C09153=1152.454,156.527,-58.181,-178.547,6.899,148.854
C09154=1152.449,156.776,-58.203,-178.545,6.901,148.853
C09155=1152.445,157.026,-58.224,-178.541,6.903,148.853
C09156=1152.440,157.274,-58.246,-178.539,6.905,148.852
C09157=1152.435,157.543,-58.269,-178.536,6.907,148.852
C09158=1152.430,157.812,-58.293,-178.533,6.909,148.852
C09159=1152.425,158.081,-58.315,-178.530,6.911,148.851
C09160=1152.420,158.351,-58.339,-178.527,6.913,148.851
C09161=1152.415,158.599,-58.360,-178.524,6.915,148.851
C09162=1152.410,158.848,-58.382,-178.521,6.917,148.850
C09163=1152.405,159.098,-58.403,-178.519,6.919,148.850
C09164=1152.400,159.346,-58.425,-178.516,6.921,148.850
C09165=1152.396,159.595,-58.447,-178.513,6.923,148.849
C09166=1152.391,159.844,-58.469,-178.510,6.925,148.849
C09167=1152.386,160.093,-58.491,-178.508,6.927,148.849
C09168=1152.382,160.343,-58.512,-178.504,6.929,148.848
C09169=1152.377,160.592,-58.534,-178.502,6.931,148.848
C09170=1152.372,160.840,-58.555,-178.499,6.933,148.848
C09171=1152.368,161.090,-58.577,-178.497,6.935,148.847
C09172=1152.363,161.338,-58.599,-178.494,6.936,148.847
C09173=1152.359,161.588,-58.621,-178.491,6.939,148.847
C09174=1152.353,161.837,-58.642,-178.488,6.941,148.846
C09175=1152.349,162.086,-58.664,-178.486,6.943,148.846
C09176=1152.344,162.335,-58.686,-178.483,6.945,148.846
C09177=1152.339,162.584,-58.707,-178.480,6.947,148.845
C09178=1152.335,162.833,-58.729,-178.477,6.949,148.845
C09179=1152.330,163.082,-58.751,-178.474,6.951,148.845
C09180=1152.326,163.331,-58.773,-178.472,6.952,148.844
C09181=1152.321,163.579,-58.795,-178.469,6.955,148.844
C09182=1152.316,163.828,-58.817,-178.466,6.957,148.844
C09183=1152.312,164.077,-58.839,-178.464,6.959,148.843
C09184=1152.307,164.326,-58.860,-178.460,6.961,148.843
C09185=1152.303,164.575,-58.882,-178.458,6.963,148.843
C09186=1152.297,164.824,-58.905,-178.455,6.965,148.842
C09187=1152.293,165.074,-58.927,-178.453,6.967,148.842
C09188=1152.288,165.322,-58.948,-178.449,6.969,148.842
C09189=1152.284,165.572,-58.970,-178.447,6.971,148.841
C09190=1152.279,165.820,-58.992,-178.444,6.973,148.841
C09191=1152.275,166.070,-59.014,-178.442,6.975,148.841
C09192=1152.270,166.318,-59.036,-178.438,6.977,148.840
C09193=1152.265,166.568,-59.058,-178.436,6.979,148.840
C09194=1152.260,166.816,-59.081,-178.433,6.981,148.840
C09195=1152.256,167.065,-59.103,-178.430,6.983,148.839
C09196=1152.251,167.314,-59.125,-178.428,6.986,148.839
C09197=1152.247,167.563,-59.147,-178.425,6.987,148.839
C09198=1152.241,167.812,-59.169,-178.422,6.989,148.838
C09199=1152.237,168.062,-59.191,-178.419,6.992,148.838
C09200=1152.233,168.310,-59.213,-178.416,6.993,148.838
C09201=1152.228,168.559,-59.235,-178.414,6.995,148.838
C09202=1152.223,168.808,-59.258,-178.411,6.998,148.837
C09203=1152.218,169.057,-59.280,-178.408,7.000,148.837
C09204=1152.214,169.307,-59.302,-178.405,7.001,148.836
C09205=1152.210,169.555,-59.324,-178.402,7.004,148.836
C09206=1152.205,169.804,-59.347,-178.400,7.006,148.836
C09207=1152.200,170.053,-59.368,-178.397,7.008,148.836
C09208=1152.195,170.302,-59.391,-178.394,7.010,148.835
C09209=1152.190,170.551,-59.413,-178.392,7.012,148.835
C09210=1152.186,170.800,-59.436,-178.389,7.014,148.835
C09211=1152.182,171.049,-59.458,-178.386,7.016,148.834
C09212=1152.176,171.298,-59.481,-178.383,7.018,148.834
C09213=1152.172,171.547,-59.503,-178.381,7.021,148.834
C09214=1152.167,171.796,-59.524,-178.378,7.022,148.833
C09215=1152.162,172.045,-59.548,-178.375,7.025,148.833
C09216=1152.158,172.294,-59.570,-178.372,7.027,148.833
C09217=1152.154,172.542,-59.592,-178.370,7.029,148.833
C09218=1152.149,172.792,-59.615,-178.366,7.031,148.832
C09219=1152.144,173.040,-59.636,-178.364,7.033,148.832
C09220=1152.139,173.289,-59.660,-178.361,7.035,148.832
C09221=1152.135,173.539,-59.682,-178.358,7.038,148.831
C09222=1152.130,173.787,-59.704,-178.356,7.039,148.831
C09223=1152.125,174.036,-59.727,-178.353,7.041,148.831
C09224=1152.121,174.285,-59.750,-178.350,7.044,148.830
C09225=1152.116,174.534,-59.772,-178.347,7.046,148.830
C09226=1152.112,174.783,-59.795,-178.345,7.047,148.830
C09227=1152.107,175.032,-59.817,-178.341,7.050,148.829
C09228=1152.102,175.280,-59.840,-178.339,7.052,148.829
C09229=1152.097,175.530,-59.862,-178.337,7.054,148.829
C09230=1152.093,175.779,-59.885,-178.333,7.056,148.829
C09231=1152.088,176.027,-59.907,-178.331,7.058,148.828
C09232=1152.084,176.276,-59.930,-178.328,7.061,148.828
C09233=1152.079,176.526,-59.952,-178.325,7.063,148.828
C09234=1152.075,176.775,-59.976,-178.322,7.065,148.827
C09235=1152.070,177.023,-59.998,-178.319,7.067,148.827
C09236=1152.065,177.272,-60.021,-178.317,7.069,148.827
C09237=1152.060,177.522,-60.044,-178.314,7.071,148.827
C09238=1152.055,177.770,-60.066,-178.311,7.073,148.826
C09239=1152.051,178.019,-60.089,-178.309,7.076,148.826
C09240=1152.047,178.268,-60.112,-178.306,7.077,148.826
C09241=1152.042,178.518,-60.134,-178.303,7.080,148.825
C09242=1152.037,178.766,-60.157,-178.300,7.082,148.825
C09243=1152.033,179.015,-60.180,-178.297,7.084,148.825
C09244=1152.029,179.263,-60.203,-178.295,7.086,148.824
C09245=1152.024,179.513,-60.226,-178.292,7.088,148.824
C09246=1152.018,179.761,-60.249,-178.289,7.091,148.824
C09247=1152.014,180.010,-60.271,-178.286,7.093,148.824
C09248=1152.010,180.259,-60.295,-178.283,7.095,148.823
C09249=1152.005,180.508,-60.317,-178.281,7.097,148.823
C09250=1152.001,180.757,-60.340,-178.278,7.099,148.823
C09251=1151.995,181.006,-60.363,-178.275,7.102,148.822
C09252=1151.991,181.255,-60.386,-178.273,7.104,148.822
C09253=1151.987,181.504,-60.409,-178.270,7.105,148.822
C09254=1151.982,181.753,-60.432,-178.267,7.108,148.822
C09255=1151.978,182.002,-60.455,-178.264,7.110,148.821
C09256=1151.973,182.251,-60.478,-178.261,7.113,148.821
C09257=1151.968,182.499,-60.501,-178.259,7.114,148.821
C09258=1151.964,182.748,-60.524,-178.256,7.116,148.821
C09259=1151.959,182.997,-60.547,-178.253,7.119,148.820
C09260=1151.954,183.246,-60.570,-178.250,7.121,148.820
C09261=1151.949,183.516,-60.596,-178.248,7.124,148.820
C09262=1151.944,183.785,-60.620,-178.244,7.126,148.819
C09263=1151.939,184.055,-60.645,-178.242,7.128,148.819
C09264=1151.934,184.325,-60.670,-178.238,7.131,148.819
C09265=1151.930,184.574,-60.693,-178.235,7.133,148.819
C09266=1151.925,184.823,-60.716,-178.233,7.135,148.818
C09267=1151.920,185.072,-60.740,-178.230,7.137,148.818
C09268=1151.916,185.321,-60.763,-178.227,7.140,148.818
C09269=1151.911,185.570,-60.786,-178.225,7.142,148.817
C09270=1151.907,185.818,-60.809,-178.221,7.144,148.817
C09271=1151.902,186.067,-60.832,-178.219,7.146,148.817
C09272=1151.897,186.315,-60.856,-178.216,7.149,148.817
C09273=1151.893,186.564,-60.879,-178.214,7.151,148.816
C09274=1151.888,186.813,-60.903,-178.211,7.153,148.816
C09275=1151.884,187.062,-60.926,-178.208,7.155,148.816
C09276=1151.879,187.311,-60.949,-178.205,7.157,148.816
C09277=1151.875,187.560,-60.972,-178.202,7.160,148.815
C09278=1151.870,187.809,-60.996,-178.200,7.162,148.815
C09279=1151.865,188.058,-61.019,-178.197,7.165,148.815
C09280=1151.860,188.307,-61.042,-178.194,7.166,148.814
C09281=1151.856,188.555,-61.066,-178.191,7.169,148.814
C09282=1151.851,188.805,-61.090,-178.189,7.171,148.814
C09283=1151.847,189.054,-61.113,-178.186,7.173,148.814
C09284=1151.843,189.302,-61.136,-178.183,7.176,148.814
C09285=1151.838,189.551,-61.159,-178.180,7.177,148.813
C09286=1151.834,189.800,-61.183,-178.178,7.180,148.813
C09287=1151.829,190.049,-61.207,-178.175,7.182,148.813
C09288=1151.824,190.298,-61.230,-178.172,7.185,148.812
C09289=1151.819,190.546,-61.253,-178.169,7.187,148.812
C09290=1151.815,190.795,-61.277,-178.166,7.189,148.812
C09291=1151.810,191.044,-61.300,-178.164,7.191,148.812
C09292=1151.805,191.293,-61.324,-178.161,7.194,148.811
C09293=1151.801,191.542,-61.348,-178.158,7.196,148.811
C09294=1151.797,191.791,-61.372,-178.155,7.199,148.811
C09295=1151.792,192.040,-61.395,-178.152,7.200,148.811
C09296=1151.787,192.289,-61.418,-178.150,7.203,148.811
C09297=1151.783,192.537,-61.442,-178.147,7.205,148.810
C09298=1151.778,192.786,-61.466,-178.145,7.207,148.810
C09299=1151.774,193.035,-61.490,-178.141,7.210,148.810
C09300=1151.769,193.284,-61.513,-178.139,7.212,148.810
C09301=1151.764,193.533,-61.537,-178.136,7.214,148.809
C09302=1151.760,193.781,-61.561,-178.133,7.216,148.809
C09303=1151.755,194.030,-61.584,-178.130,7.219,148.809
C09304=1151.750,194.279,-61.609,-178.128,7.221,148.808
C09305=1151.745,194.528,-61.632,-178.125,7.224,148.808
C09306=1151.741,194.776,-61.656,-178.122,7.225,148.808
C09307=1151.736,195.025,-61.679,-178.120,7.228,148.808
C09308=1151.732,195.274,-61.704,-178.117,7.230,148.807
C09309=1151.727,195.523,-61.727,-178.114,7.233,148.807
C09310=1151.723,195.771,-61.751,-178.111,7.235,148.807
C09311=1151.719,196.021,-61.775,-178.109,7.238,148.807
C09312=1151.714,196.269,-61.799,-178.106,7.239,148.807
C09313=1151.709,196.519,-61.823,-178.103,7.242,148.806
C09314=1151.705,196.767,-61.847,-178.100,7.244,148.806
C09315=1151.700,197.016,-61.870,-178.097,7.247,148.806
C09316=1151.695,197.265,-61.894,-178.094,7.250,148.806
C09317=1151.691,197.513,-61.918,-178.092,7.251,148.805
C09318=1151.687,197.763,-61.942,-178.089,7.254,148.805
C09319=1151.682,198.011,-61.967,-178.086,7.256,148.805
C09320=1151.677,198.260,-61.991,-178.083,7.259,148.805
C09321=1151.673,198.509,-62.014,-178.081,7.261,148.804
C09322=1151.668,198.757,-62.038,-178.078,7.264,148.804
C09323=1151.663,199.006,-62.063,-178.075,7.265,148.804
C09324=1151.659,199.255,-62.086,-178.072,7.268,148.804
C09325=1151.655,199.504,-62.111,-178.070,7.270,148.803
C09326=1151.650,199.753,-62.135,-178.067,7.273,148.803
C09327=1151.645,200.002,-62.159,-178.064,7.275,148.803
C09328=1151.640,200.250,-62.183,-178.061,7.278,148.803
C09329=1151.636,200.499,-62.207,-178.059,7.279,148.803
C09330=1151.632,200.748,-62.231,-178.056,7.282,148.802
C09331=1151.627,200.997,-62.256,-178.053,7.285,148.802
C09332=1151.622,201.246,-62.279,-178.050,7.287,148.802
C09333=1151.618,201.494,-62.303,-178.047,7.289,148.802
C09334=1151.614,201.743,-62.328,-178.045,7.292,148.802
C09335=1151.609,201.992,-62.353,-178.042,7.294,148.801
C09336=1151.605,202.240,-62.377,-178.040,7.296,148.801
C09337=1151.600,202.489,-62.401,-178.036,7.299,148.801
C09338=1151.596,202.739,-62.425,-178.034,7.301,148.801
C09339=1151.591,202.987,-62.449,-178.031,7.303,148.800
C09340=1151.586,203.236,-62.474,-178.028,7.306,148.800
C09341=1151.582,203.484,-62.498,-178.025,7.308,148.800
C09342=1151.578,203.733,-62.522,-178.023,7.311,148.800
C09343=1151.573,203.982,-62.547,-178.020,7.313,148.799
C09344=1151.568,204.231,-62.571,-178.017,7.316,148.799
C09345=1151.563,204.479,-62.596,-178.015,7.318,148.799
C09346=1151.559,204.728,-62.620,-178.012,7.320,148.799
C09347=1151.554,204.977,-62.645,-178.009,7.323,148.799
C09348=1151.550,205.226,-62.669,-178.006,7.325,148.798
C09349=1151.546,205.475,-62.693,-178.003,7.328,148.798
C09350=1151.541,205.723,-62.718,-178.001,7.330,148.798
C09351=1151.537,205.972,-62.742,-177.998,7.333,148.798
C09352=1151.532,206.221,-62.767,-177.995,7.334,148.797
C09353=1151.528,206.470,-62.791,-177.992,7.337,148.797
C09354=1151.522,206.718,-62.816,-177.989,7.340,148.797
C09355=1151.518,206.967,-62.840,-177.987,7.342,148.797
C09356=1151.514,207.216,-62.865,-177.984,7.345,148.797
C09357=1151.509,207.465,-62.889,-177.981,7.347,148.796
C09358=1151.505,207.714,-62.914,-177.979,7.350,148.796
C09359=1151.501,207.962,-62.939,-177.975,7.352,148.796
C09360=1151.495,208.211,-62.963,-177.973,7.354,148.796
C09361=1151.491,208.460,-62.989,-177.970,7.357,148.796
C09362=1151.486,208.708,-63.013,-177.968,7.359,148.795
C09363=1151.481,208.957,-63.037,-177.965,7.362,148.795
C09364=1151.478,209.206,-63.062,-177.962,7.364,148.795
C09365=1151.472,209.476,-63.088,-177.959,7.367,148.795
C09366=1151.468,209.747,-63.115,-177.956,7.369,148.795
C09367=1151.462,210.018,-63.143,-177.953,7.372,148.795
C09368=1151.457,210.289,-63.170,-177.950,7.375,148.794
C09369=1151.453,210.536,-63.195,-177.947,7.378,148.794
C09370=1151.448,210.785,-63.219,-177.944,7.380,148.794
C09371=1151.444,211.034,-63.244,-177.942,7.382,148.794
C09372=1151.439,211.283,-63.268,-177.939,7.385,148.794
C09373=1151.435,211.532,-63.294,-177.936,7.387,148.793
C09374=1151.431,211.780,-63.318,-177.934,7.390,148.793
C09375=1151.426,212.030,-63.343,-177.930,7.392,148.793
C09376=1151.421,212.278,-63.369,-177.928,7.394,148.793
C09377=1151.417,212.527,-63.393,-177.925,7.397,148.793
C09378=1151.412,212.776,-63.418,-177.922,7.400,148.792
C09379=1151.408,213.024,-63.443,-177.920,7.402,148.792
C09380=1151.403,213.273,-63.468,-177.917,7.405,148.792
C09381=1151.399,213.521,-63.493,-177.914,7.408,148.792
C09382=1151.394,213.770,-63.518,-177.912,7.410,148.792
C09383=1151.390,214.018,-63.543,-177.908,7.412,148.791
C09384=1151.385,214.268,-63.568,-177.906,7.414,148.791
C09385=1151.381,214.516,-63.593,-177.903,7.417,148.791
C09386=1151.376,214.765,-63.618,-177.900,7.420,148.791
C09387=1151.371,215.014,-63.643,-177.898,7.422,148.791
C09388=1151.367,215.263,-63.669,-177.895,7.425,148.791
C09389=1151.363,215.510,-63.694,-177.892,7.427,148.790
C09390=1151.358,215.760,-63.719,-177.890,7.430,148.790
C09391=1151.354,216.008,-63.744,-177.886,7.432,148.790
C09392=1151.349,216.257,-63.769,-177.884,7.435,148.790
C09393=1151.345,216.506,-63.795,-177.881,7.437,148.790
C09394=1151.340,216.755,-63.819,-177.878,7.440,148.789
C09395=1151.336,217.003,-63.845,-177.875,7.443,148.789
C09396=1151.331,217.252,-63.869,-177.873,7.445,148.789
C09397=1151.327,217.501,-63.895,-177.870,7.447,148.789
C09398=1151.322,217.749,-63.920,-177.867,7.450,148.789
C09399=1151.318,217.998,-63.945,-177.865,7.452,148.789
C09400=1151.313,218.246,-63.971,-177.862,7.455,148.788
C09401=1151.309,218.495,-63.996,-177.859,7.458,148.788
C09402=1151.305,218.744,-64.021,-177.857,7.460,148.788
C09403=1151.300,218.992,-64.046,-177.853,7.463,148.788
C09404=1151.296,219.241,-64.072,-177.851,7.466,148.788
C09405=1151.291,219.489,-64.097,-177.848,7.468,148.788
C09406=1151.286,219.739,-64.123,-177.845,7.470,148.787
C09407=1151.282,219.988,-64.148,-177.842,7.473,148.787
C09408=1151.277,220.236,-64.174,-177.839,7.476,148.787
C09409=1151.273,220.485,-64.199,-177.837,7.478,148.787
C09410=1151.268,220.734,-64.224,-177.834,7.481,148.787
C09411=1151.264,220.982,-64.250,-177.831,7.484,148.786
C09412=1151.259,221.231,-64.276,-177.829,7.486,148.786
C09413=1151.255,221.479,-64.301,-177.826,7.488,148.786
C09414=1151.250,221.728,-64.327,-177.823,7.491,148.786
C09415=1151.246,221.977,-64.352,-177.820,7.494,148.786
C09416=1151.241,222.225,-64.377,-177.818,7.496,148.786
C09417=1151.237,222.474,-64.403,-177.815,7.499,148.785
C09418=1151.233,222.723,-64.429,-177.812,7.502,148.785
C09419=1151.228,222.971,-64.454,-177.810,7.504,148.785
C09420=1151.223,223.220,-64.480,-177.806,7.506,148.785
C09421=1151.219,223.469,-64.506,-177.804,7.509,148.785
C09422=1151.214,223.717,-64.531,-177.801,7.512,148.785
C09423=1151.210,223.966,-64.557,-177.799,7.514,148.785
C09424=1151.206,224.214,-64.582,-177.795,7.517,148.784
C09425=1151.202,224.463,-64.608,-177.793,7.520,148.784
C09426=1151.197,224.711,-64.634,-177.790,7.523,148.784
C09427=1151.193,224.960,-64.659,-177.787,7.525,148.784
C09428=1151.188,225.209,-64.686,-177.784,7.528,148.784
C09429=1151.183,225.457,-64.711,-177.782,7.530,148.784
C09430=1151.179,225.706,-64.737,-177.779,7.533,148.784
C09431=1151.174,225.955,-64.763,-177.776,7.535,148.783
C09432=1151.170,226.204,-64.788,-177.773,7.538,148.783
C09433=1151.165,226.452,-64.814,-177.771,7.541,148.783
C09434=1151.161,226.701,-64.839,-177.768,7.543,148.783
C09435=1151.156,226.950,-64.866,-177.765,7.546,148.783
C09436=1151.152,227.199,-64.892,-177.762,7.549,148.783
C09437=1151.148,227.446,-64.918,-177.760,7.552,148.782
C09438=1151.143,227.695,-64.943,-177.757,7.555,148.782
C09439=1151.139,227.944,-64.969,-177.754,7.556,148.782
C09440=1151.134,228.193,-64.995,-177.751,7.559,148.782
C09441=1151.130,228.442,-65.021,-177.749,7.562,148.782
C09442=1151.125,228.690,-65.047,-177.746,7.565,148.782
C09443=1151.121,228.938,-65.073,-177.743,7.567,148.781
C09444=1151.116,229.187,-65.099,-177.740,7.570,148.781
C09445=1151.112,229.436,-65.125,-177.737,7.573,148.781
C09446=1151.108,229.685,-65.151,-177.735,7.576,148.781
C09447=1151.103,229.932,-65.177,-177.732,7.578,148.781
C09448=1151.098,230.181,-65.203,-177.729,7.580,148.781
C09449=1151.094,230.430,-65.229,-177.726,7.583,148.781
C09450=1151.090,230.679,-65.255,-177.724,7.586,148.781
C09451=1151.085,230.927,-65.282,-177.721,7.589,148.781
C09452=1151.081,231.176,-65.308,-177.719,7.591,148.780
C09453=1151.076,231.424,-65.333,-177.715,7.594,148.780
C09454=1151.071,231.673,-65.360,-177.713,7.597,148.780
C09455=1151.067,231.921,-65.386,-177.710,7.600,148.780
C09456=1151.063,232.170,-65.412,-177.708,7.602,148.780
C09457=1151.058,232.419,-65.439,-177.705,7.605,148.780
C09458=1151.054,232.668,-65.464,-177.702,7.607,148.779
C09459=1151.050,232.916,-65.491,-177.699,7.610,148.779
C09460=1151.045,233.165,-65.517,-177.696,7.613,148.779
C09461=1151.041,233.412,-65.543,-177.694,7.615,148.779
C09462=1151.036,233.661,-65.570,-177.691,7.618,148.779
C09463=1151.032,233.910,-65.596,-177.688,7.621,148.779
C09464=1151.028,234.158,-65.622,-177.685,7.624,148.779
C09465=1151.023,234.407,-65.649,-177.682,7.627,148.779
C09466=1151.019,234.656,-65.675,-177.680,7.629,148.779
C09467=1151.014,234.904,-65.702,-177.677,7.632,148.778
C09468=1151.010,235.153,-65.728,-177.674,7.635,148.778
C09469=1151.005,235.425,-65.757,-177.671,7.637,148.778
C09470=1151.000,235.697,-65.785,-177.668,7.640,148.778
C09471=1150.995,235.968,-65.814,-177.665,7.644,148.778
C09472=1150.990,236.240,-65.844,-177.662,7.646,148.778
C09473=1150.986,236.489,-65.869,-177.659,7.649,148.778
C09474=1150.981,236.737,-65.896,-177.657,7.651,148.777
C09475=1150.977,236.985,-65.923,-177.654,7.654,148.777
C09476=1150.972,237.234,-65.949,-177.651,7.657,148.777
C09477=1150.968,237.483,-65.976,-177.648,7.660,148.777
C09478=1150.963,237.731,-66.003,-177.646,7.663,148.777
C09479=1150.959,237.980,-66.029,-177.642,7.666,148.777
C09480=1150.955,238.228,-66.056,-177.640,7.668,148.777
C09481=1150.951,238.477,-66.082,-177.637,7.671,148.777
C09482=1150.946,238.726,-66.108,-177.635,7.674,148.777
C09483=1150.941,238.974,-66.135,-177.632,7.677,148.777
C09484=1150.937,239.222,-66.162,-177.629,7.680,148.776
C09485=1150.932,239.471,-66.189,-177.626,7.683,148.776
C09486=1150.928,239.719,-66.215,-177.624,7.684,148.776
C09487=1150.924,239.968,-66.242,-177.621,7.687,148.776
C09488=1150.919,240.217,-66.269,-177.618,7.690,148.776
C09489=1150.916,240.465,-66.296,-177.615,7.693,148.776
C09490=1150.911,240.714,-66.323,-177.613,7.696,148.776
C09491=1150.906,240.962,-66.350,-177.610,7.699,148.776
C09492=1150.902,241.211,-66.376,-177.607,7.702,148.776
C09493=1150.897,241.460,-66.403,-177.605,7.704,148.775
C09494=1150.893,241.708,-66.430,-177.602,7.707,148.775
C09495=1150.889,241.956,-66.456,-177.599,7.710,148.775
C09496=1150.884,242.205,-66.483,-177.596,7.712,148.775
C09497=1150.879,242.453,-66.510,-177.593,7.715,148.775
C09498=1150.876,242.702,-66.537,-177.590,7.718,148.775
C09499=1150.871,242.950,-66.564,-177.588,7.721,148.775
C09500=1150.866,243.199,-66.591,-177.585,7.723,148.775
C09501=1150.862,243.448,-66.618,-177.583,7.726,148.775
C09502=1150.858,243.696,-66.645,-177.580,7.729,148.775
C09503=1150.854,243.944,-66.672,-177.577,7.732,148.774
C09504=1150.849,244.193,-66.699,-177.574,7.735,148.774
C09505=1150.844,244.441,-66.726,-177.571,7.738,148.774
C09506=1150.840,244.690,-66.753,-177.568,7.741,148.774
C09507=1150.836,244.938,-66.779,-177.565,7.744,148.774
C09508=1150.831,245.187,-66.807,-177.563,7.746,148.774
C09509=1150.827,245.436,-66.834,-177.560,7.749,148.774
C09510=1150.822,245.684,-66.861,-177.558,7.751,148.774
C09511=1150.818,245.933,-66.888,-177.555,7.754,148.774
C09512=1150.814,246.180,-66.915,-177.552,7.757,148.774
C09513=1150.809,246.429,-66.942,-177.549,7.760,148.774
C09514=1150.805,246.678,-66.970,-177.547,7.763,148.773
C09515=1150.801,246.927,-66.997,-177.544,7.766,148.773
C09516=1150.796,247.175,-67.024,-177.541,7.769,148.773
C09517=1150.791,247.424,-67.051,-177.539,7.771,148.773
C09518=1150.787,247.671,-67.079,-177.536,7.774,148.773
C09519=1150.782,247.920,-67.106,-177.533,7.777,148.773
C09520=1150.778,248.169,-67.133,-177.530,7.780,148.773
C09521=1150.774,248.417,-67.160,-177.528,7.783,148.773
C09522=1150.770,248.665,-67.187,-177.525,7.786,148.773
C09523=1150.765,248.914,-67.215,-177.522,7.789,148.773
C09524=1150.761,249.163,-67.242,-177.519,7.792,148.773
C09525=1150.757,249.411,-67.269,-177.517,7.795,148.773
C09526=1150.752,249.659,-67.297,-177.513,7.797,148.772
C09527=1150.748,249.908,-67.324,-177.511,7.799,148.772
C09528=1150.744,250.157,-67.351,-177.508,7.802,148.772
C09529=1150.739,250.405,-67.379,-177.506,7.805,148.772
C09530=1150.735,250.653,-67.406,-177.503,7.808,148.772
C09531=1150.730,250.901,-67.434,-177.500,7.811,148.772
C09532=1150.726,251.150,-67.461,-177.497,7.814,148.772
C09533=1150.722,251.399,-67.488,-177.494,7.817,148.772
C09534=1150.717,251.647,-67.516,-177.492,7.820,148.772
C09535=1150.713,251.896,-67.544,-177.489,7.823,148.772
C09536=1150.709,252.144,-67.571,-177.486,7.826,148.772
C09537=1150.704,252.392,-67.598,-177.483,7.829,148.772
C09538=1150.700,252.640,-67.626,-177.481,7.832,148.771
C09539=1150.696,252.889,-67.654,-177.478,7.835,148.771
C09540=1150.691,253.138,-67.682,-177.475,7.838,148.771
C09541=1150.686,253.386,-67.709,-177.473,7.840,148.771
C09542=1150.682,253.635,-67.737,-177.470,7.843,148.771
C09543=1150.678,253.883,-67.764,-177.467,7.845,148.771
C09544=1150.673,254.131,-67.792,-177.464,7.848,148.771
C09545=1150.669,254.380,-67.819,-177.462,7.851,148.771
C09546=1150.665,254.628,-67.847,-177.459,7.855,148.771
C09547=1150.661,254.877,-67.875,-177.457,7.858,148.771
C09548=1150.656,255.126,-67.903,-177.454,7.860,148.771
C09549=1150.651,255.373,-67.931,-177.451,7.863,148.771
C09550=1150.647,255.623,-67.958,-177.448,7.866,148.771
C09551=1150.643,255.870,-67.986,-177.445,7.869,148.771
C09552=1150.639,256.118,-68.014,-177.443,7.872,148.771
C09553=1150.635,256.368,-68.041,-177.440,7.875,148.771
C09554=1150.629,256.616,-68.070,-177.437,7.878,148.771
C09555=1150.626,256.864,-68.098,-177.434,7.881,148.771
C09556=1150.621,257.113,-68.125,-177.432,7.884,148.770
C09557=1150.617,257.361,-68.153,-177.429,7.887,148.770
C09558=1150.612,257.610,-68.181,-177.426,7.890,148.770
C09559=1150.608,257.857,-68.209,-177.423,7.893,148.770
C09560=1150.604,258.107,-68.237,-177.420,7.896,148.770
C09561=1150.599,258.355,-68.264,-177.418,7.899,148.770
C09562=1150.595,258.603,-68.293,-177.415,7.901,148.770
C09563=1150.591,258.851,-68.321,-177.413,7.904,148.770
C09564=1150.586,259.099,-68.349,-177.410,7.907,148.770
C09565=1150.581,259.349,-68.377,-177.408,7.910,148.770
C09566=1150.577,259.597,-68.404,-177.405,7.913,148.770
C09567=1150.573,259.845,-68.433,-177.402,7.916,148.770
C09568=1150.568,260.093,-68.461,-177.399,7.919,148.770
C09569=1150.565,260.342,-68.489,-177.396,7.922,148.770
C09570=1150.560,260.590,-68.517,-177.394,7.925,148.770
C09571=1150.556,260.839,-68.546,-177.391,7.928,148.770
C09572=1150.551,261.087,-68.573,-177.388,7.930,148.770
C09573=1150.547,261.360,-68.604,-177.385,7.934,148.770
C09574=1150.542,261.633,-68.635,-177.382,7.937,148.770
C09575=1150.537,261.907,-68.666,-177.379,7.940,148.770
C09576=1150.533,262.181,-68.697,-177.376,7.944,148.769
C09577=1150.528,262.429,-68.725,-177.373,7.947,148.769
C09578=1150.524,262.678,-68.754,-177.370,7.950,148.769
C09579=1150.520,262.925,-68.782,-177.368,7.953,148.770
C09580=1150.515,263.174,-68.811,-177.365,7.956,148.769
C09581=1150.511,263.422,-68.839,-177.362,7.959,148.769
C09582=1150.506,263.671,-68.867,-177.360,7.962,148.769
C09583=1150.502,263.918,-68.895,-177.357,7.965,148.769
C09584=1150.497,264.167,-68.924,-177.354,7.968,148.769
C09585=1150.493,264.415,-68.952,-177.351,7.971,148.769
C09586=1150.489,264.664,-68.980,-177.349,7.974,148.769
C09587=1150.485,264.913,-69.008,-177.346,7.977,148.769
C09588=1150.480,265.161,-69.037,-177.343,7.980,148.769
C09589=1150.476,265.409,-69.066,-177.341,7.983,148.769
C09590=1150.471,265.657,-69.094,-177.338,7.986,148.769
C09591=1150.468,265.906,-69.122,-177.335,7.989,148.769
C09592=1150.463,266.154,-69.151,-177.332,7.991,148.769
C09593=1150.459,266.402,-69.179,-177.330,7.995,148.769
C09594=1150.455,266.651,-69.208,-177.327,7.998,148.769
C09595=1150.449,266.899,-69.237,-177.324,8.001,148.769
C09596=1150.446,267.147,-69.265,-177.322,8.004,148.769
C09597=1150.441,267.396,-69.293,-177.319,8.007,148.769
C09598=1150.437,267.643,-69.322,-177.316,8.009,148.769
C09599=1150.433,267.892,-69.351,-177.314,8.013,148.769
C09600=1150.428,268.141,-69.379,-177.311,8.016,148.769
C09601=1150.424,268.388,-69.408,-177.308,8.019,148.769
C09602=1150.420,268.637,-69.437,-177.305,8.022,148.769
C09603=1150.415,268.885,-69.464,-177.303,8.024,148.769
C09604=1150.411,269.134,-69.494,-177.300,8.027,148.769
C09605=1150.407,269.382,-69.523,-177.298,8.031,148.769
C09606=1150.403,269.630,-69.551,-177.295,8.034,148.769
C09607=1150.398,269.879,-69.580,-177.292,8.037,148.769
C09608=1150.394,270.127,-69.609,-177.289,8.040,148.769
C09609=1150.390,270.375,-69.637,-177.286,8.042,148.769
C09610=1150.385,270.624,-69.666,-177.284,8.047,148.769
C09611=1150.381,270.872,-69.695,-177.281,8.049,148.769
C09612=1150.376,271.121,-69.724,-177.278,8.052,148.769
C09613=1150.372,271.368,-69.752,-177.275,8.055,148.769
C09614=1150.368,271.617,-69.781,-177.273,8.059,148.769
C09615=1150.364,271.865,-69.811,-177.270,8.062,148.769
C09616=1150.359,272.114,-69.839,-177.267,8.064,148.769
C09617=1150.355,272.361,-69.868,-177.265,8.067,148.769
C09618=1150.351,272.610,-69.897,-177.262,8.070,148.769
C09619=1150.346,272.858,-69.926,-177.260,8.074,148.769
C09620=1150.342,273.107,-69.956,-177.257,8.077,148.769
C09621=1150.338,273.355,-69.983,-177.254,8.080,148.769
C09622=1150.334,273.603,-70.013,-177.251,8.082,148.769
C09623=1150.329,273.852,-70.041,-177.249,8.086,148.769
C09624=1150.325,274.100,-70.071,-177.246,8.089,148.769
C09625=1150.320,274.348,-70.100,-177.243,8.092,148.769
C09626=1150.316,274.596,-70.129,-177.241,8.095,148.769
C09627=1150.312,274.844,-70.158,-177.238,8.099,148.769
C09628=1150.308,275.093,-70.187,-177.235,8.102,148.769
C09629=1150.304,275.341,-70.217,-177.232,8.105,148.769
C09630=1150.299,275.589,-70.245,-177.229,8.107,148.769
C09631=1150.295,275.837,-70.274,-177.227,8.111,148.769
C09632=1150.291,276.086,-70.304,-177.224,8.114,148.769
C09633=1150.286,276.334,-70.333,-177.221,8.117,148.769
C09634=1150.282,276.583,-70.362,-177.219,8.120,148.769
C09635=1150.278,276.831,-70.391,-177.216,8.123,148.769
C09636=1150.274,277.078,-70.420,-177.214,8.126,148.769
C09637=1150.269,277.327,-70.449,-177.211,8.129,148.769
C09638=1150.265,277.575,-70.479,-177.208,8.132,148.769
C09639=1150.261,277.824,-70.508,-177.206,8.135,148.769
C09640=1150.257,278.072,-70.537,-177.202,8.139,148.769
C09641=1150.252,278.320,-70.566,-177.200,8.142,148.769
C09642=1150.248,278.569,-70.596,-177.197,8.145,148.769
C09643=1150.244,278.817,-70.625,-177.194,8.148,148.769
C09644=1150.239,279.064,-70.654,-177.192,8.151,148.769
C09645=1150.235,279.313,-70.684,-177.189,8.154,148.769
C09646=1150.231,279.561,-70.713,-177.187,8.157,148.769
C09647=1150.227,279.809,-70.743,-177.184,8.160,148.769
C09648=1150.223,280.057,-70.772,-177.182,8.163,148.769
C09649=1150.218,280.306,-70.802,-177.179,8.166,148.769
C09650=1150.214,280.554,-70.831,-177.175,8.170,148.769
C09651=1150.210,280.802,-70.861,-177.173,8.173,148.769
C09652=1150.206,281.051,-70.890,-177.170,8.176,148.769
C09653=1150.201,281.299,-70.920,-177.168,8.179,148.769
C09654=1150.197,281.547,-70.950,-177.165,8.182,148.769
C09655=1150.192,281.795,-70.979,-177.162,8.185,148.769
C09656=1150.188,282.043,-71.008,-177.160,8.189,148.769
C09657=1150.184,282.292,-71.038,-177.157,8.191,148.769
C09658=1150.179,282.540,-71.067,-177.155,8.194,148.769
C09659=1150.175,282.788,-71.097,-177.152,8.198,148.770
C09660=1150.171,283.036,-71.127,-177.149,8.201,148.770
C09661=1150.166,283.284,-71.157,-177.146,8.204,148.769
C09662=1150.162,283.533,-71.186,-177.144,8.208,148.770
C09663=1150.158,283.781,-71.216,-177.141,8.211,148.770
C09664=1150.154,284.029,-71.245,-177.138,8.214,148.770
C09665=1150.150,284.277,-71.275,-177.136,8.217,148.770
C09666=1150.145,284.525,-71.305,-177.133,8.220,148.770
C09667=1150.141,284.774,-71.335,-177.130,8.224,148.770
C09668=1150.137,285.022,-71.364,-177.127,8.227,148.770
C09669=1150.133,285.270,-71.394,-177.125,8.230,148.770
C09670=1150.129,285.518,-71.424,-177.122,8.233,148.770
C09671=1150.124,285.766,-71.454,-177.120,8.236,148.770
C09672=1150.120,286.015,-71.483,-177.117,8.239,148.770
C09673=1150.116,286.262,-71.514,-177.115,8.242,148.770
C09674=1150.112,286.511,-71.543,-177.111,8.246,148.770
C09675=1150.107,286.759,-71.573,-177.109,8.249,148.770
C09676=1150.103,287.007,-71.603,-177.106,8.252,148.770
C09677=1150.098,287.283,-71.636,-177.104,8.255,148.770
C09678=1150.094,287.558,-71.669,-177.100,8.259,148.770
C09679=1150.089,287.833,-71.702,-177.097,8.263,148.770
C09680=1150.084,288.109,-71.736,-177.095,8.266,148.770
C09681=1150.080,288.357,-71.766,-177.092,8.269,148.770
C09682=1150.076,288.605,-71.796,-177.089,8.273,148.770
C09683=1150.071,288.853,-71.826,-177.086,8.276,148.771
C09684=1150.067,289.101,-71.856,-177.084,8.279,148.771
C09685=1150.063,289.349,-71.886,-177.081,8.282,148.771
C09686=1150.058,289.597,-71.916,-177.078,8.285,148.771
C09687=1150.054,289.845,-71.946,-177.076,8.289,148.771
C09688=1150.050,290.094,-71.977,-177.073,8.292,148.771
C09689=1150.046,290.342,-72.007,-177.070,8.296,148.771
C09690=1150.042,290.590,-72.037,-177.068,8.299,148.771
C09691=1150.038,290.838,-72.067,-177.065,8.302,148.771
C09692=1150.033,291.086,-72.097,-177.063,8.305,148.771
C09693=1150.029,291.334,-72.128,-177.060,8.308,148.771
C09694=1150.025,291.582,-72.157,-177.057,8.312,148.771
C09695=1150.021,291.831,-72.188,-177.054,8.315,148.771
C09696=1150.017,292.079,-72.218,-177.052,8.318,148.771
C09697=1150.012,292.327,-72.248,-177.049,8.321,148.771
C09698=1150.008,292.575,-72.279,-177.047,8.324,148.772
C09699=1150.004,292.823,-72.309,-177.044,8.327,148.772
C09700=1150.000,293.071,-72.340,-177.041,8.331,148.772
C09701=1149.996,293.320,-72.369,-177.038,8.334,148.772
C09702=1149.991,293.567,-72.400,-177.036,8.337,148.772
C09703=1149.987,293.815,-72.431,-177.033,8.340,148.772
C09704=1149.982,294.064,-72.460,-177.031,8.344,148.772
C09705=1149.978,294.312,-72.491,-177.028,8.347,148.772
C09706=1149.974,294.560,-72.522,-177.025,8.351,148.772
C09707=1149.970,294.808,-72.552,-177.022,8.354,148.772
C09708=1149.966,295.056,-72.583,-177.020,8.357,148.772
C09709=1149.962,295.305,-72.613,-177.017,8.360,148.772
C09710=1149.958,295.553,-72.643,-177.014,8.364,148.773
C09711=1149.953,295.801,-72.674,-177.012,8.367,148.773
C09712=1149.949,296.048,-72.705,-177.009,8.370,148.773
C09713=1149.945,296.297,-72.735,-177.007,8.373,148.773
C09714=1149.941,296.545,-72.766,-177.004,8.376,148.773
C09715=1149.937,296.792,-72.796,-177.001,8.381,148.773
C09716=1149.932,297.040,-72.827,-176.999,8.383,148.773
C09717=1149.928,297.289,-72.858,-176.996,8.387,148.773
C09718=1149.924,297.537,-72.888,-176.993,8.390,148.773
C09719=1149.920,297.785,-72.919,-176.991,8.393,148.773
C09720=1149.916,298.033,-72.950,-176.988,8.397,148.773
C09721=1149.912,298.281,-72.980,-176.985,8.400,148.773
C09722=1149.907,298.529,-73.011,-176.983,8.403,148.774
C09723=1149.903,298.777,-73.042,-176.980,8.406,148.774
C09724=1149.899,299.026,-73.073,-176.978,8.410,148.774
C09725=1149.895,299.273,-73.103,-176.975,8.413,148.774
C09726=1149.890,299.521,-73.134,-176.972,8.417,148.774
C09727=1149.886,299.770,-73.165,-176.970,8.420,148.774
C09728=1149.881,300.018,-73.196,-176.967,8.423,148.774
C09729=1149.878,300.265,-73.226,-176.964,8.427,148.774
C09730=1149.874,300.514,-73.257,-176.962,8.430,148.774
C09731=1149.869,300.762,-73.288,-176.959,8.433,148.774
C09732=1149.865,301.011,-73.319,-176.957,8.436,148.775
C09733=1149.861,301.258,-73.350,-176.954,8.440,148.775
C09734=1149.857,301.506,-73.381,-176.951,8.443,148.775
C09735=1149.853,301.754,-73.412,-176.949,8.446,148.775
C09736=1149.848,302.002,-73.442,-176.946,8.450,148.775
C09737=1149.844,302.250,-73.473,-176.943,8.454,148.775
C09738=1149.840,302.498,-73.505,-176.941,8.457,148.775
C09739=1149.836,302.746,-73.535,-176.938,8.460,148.775
C09740=1149.832,302.995,-73.566,-176.936,8.463,148.776
C09741=1149.827,303.243,-73.597,-176.933,8.466,148.776
C09742=1149.823,303.490,-73.629,-176.930,8.470,148.776
C09743=1149.819,303.739,-73.660,-176.927,8.473,148.776
C09744=1149.814,303.986,-73.690,-176.925,8.476,148.776
C09745=1149.811,304.235,-73.722,-176.923,8.480,148.776
C09746=1149.806,304.482,-73.753,-176.920,8.483,148.776
C09747=1149.802,304.731,-73.784,-176.917,8.487,148.776
C09748=1149.798,304.978,-73.816,-176.915,8.490,148.776
C09749=1149.793,305.226,-73.846,-176.912,8.494,148.776
C09750=1149.789,305.474,-73.878,-176.909,8.497,148.777
C09751=1149.785,305.722,-73.909,-176.907,8.500,148.777
C09752=1149.782,305.971,-73.940,-176.904,8.503,148.777
C09753=1149.777,306.218,-73.971,-176.901,8.507,148.777
C09754=1149.773,306.467,-74.002,-176.899,8.511,148.777
C09755=1149.769,306.714,-74.034,-176.896,8.514,148.777
C09756=1149.765,306.963,-74.065,-176.894,8.517,148.777
C09757=1149.761,307.210,-74.096,-176.891,8.521,148.778
C09758=1149.756,307.459,-74.128,-176.889,8.524,148.778
C09759=1149.752,307.706,-74.160,-176.886,8.527,148.778
C09760=1149.748,307.955,-74.191,-176.883,8.530,148.778
C09761=1149.743,308.202,-74.222,-176.881,8.534,148.778
C09762=1149.739,308.451,-74.253,-176.878,8.537,148.778
C09763=1149.735,308.698,-74.285,-176.875,8.541,148.778
C09764=1149.731,308.946,-74.317,-176.873,8.545,148.778
C09765=1149.727,309.194,-74.347,-176.870,8.548,148.779
C09766=1149.723,309.442,-74.379,-176.867,8.551,148.779
C09767=1149.719,309.690,-74.411,-176.865,8.554,148.779
C09768=1149.715,309.938,-74.442,-176.862,8.558,148.779
C09769=1149.711,310.186,-74.474,-176.859,8.561,148.779
C09770=1149.706,310.434,-74.506,-176.857,8.565,148.779
C09771=1149.702,310.683,-74.537,-176.854,8.569,148.779
C09772=1149.697,310.930,-74.568,-176.852,8.572,148.780
C09773=1149.694,311.178,-74.600,-176.849,8.575,148.780
C09774=1149.689,311.426,-74.631,-176.846,8.579,148.780
C09775=1149.685,311.674,-74.663,-176.844,8.582,148.780
C09776=1149.682,311.922,-74.695,-176.842,8.586,148.780
C09777=1149.677,312.170,-74.727,-176.839,8.588,148.780
C09778=1149.673,312.418,-74.759,-176.836,8.593,148.780
C09779=1149.668,312.666,-74.789,-176.834,8.596,148.781
C09780=1149.665,312.914,-74.821,-176.831,8.599,148.781
C09781=1149.660,313.191,-74.857,-176.828,8.603,148.781
C09782=1149.655,313.469,-74.893,-176.825,8.607,148.781
C09783=1149.651,313.747,-74.929,-176.822,8.611,148.781
C09784=1149.646,314.024,-74.964,-176.819,8.615,148.781
C09785=1149.642,314.272,-74.996,-176.817,8.618,148.782
C09786=1149.638,314.521,-75.027,-176.814,8.621,148.782
C09787=1149.633,314.768,-75.059,-176.811,8.625,148.782
C09788=1149.630,315.016,-75.091,-176.809,8.629,148.782
C09789=1149.625,315.264,-75.123,-176.807,8.632,148.782
C09790=1149.621,315.512,-75.155,-176.804,8.636,148.782
C09791=1149.617,315.760,-75.186,-176.801,8.639,148.783
C09792=1149.613,316.008,-75.218,-176.799,8.642,148.783
C09793=1149.609,316.256,-75.251,-176.796,8.646,148.783
C09794=1149.605,316.503,-75.282,-176.793,8.650,148.783
C09795=1149.600,316.752,-75.315,-176.791,8.653,148.783
C09796=1149.597,317.000,-75.347,-176.788,8.657,148.783
C09797=1149.593,317.247,-75.379,-176.786,8.660,148.784
C09798=1149.588,317.495,-75.411,-176.783,8.663,148.784
C09799=1149.584,317.743,-75.443,-176.780,8.667,148.784
C09800=1149.581,317.991,-75.475,-176.778,8.671,148.784
C09801=1149.576,318.239,-75.507,-176.776,8.674,148.784
C09802=1149.572,318.487,-75.539,-176.773,8.678,148.784
C09803=1149.567,318.735,-75.571,-176.770,8.681,148.785
C09804=1149.564,318.983,-75.603,-176.768,8.684,148.785
C09805=1149.560,319.230,-75.635,-176.765,8.688,148.785
C09806=1149.555,319.478,-75.668,-176.762,8.692,148.785
C09807=1149.552,319.726,-75.700,-176.760,8.695,148.785
C09808=1149.547,319.975,-75.732,-176.757,8.699,148.785
C09809=1149.544,320.222,-75.765,-176.755,8.702,148.786
C09810=1149.539,320.470,-75.797,-176.752,8.705,148.786
C09811=1149.535,320.718,-75.828,-176.750,8.710,148.786
C09812=1149.531,320.966,-75.861,-176.747,8.713,148.786
C09813=1149.527,321.213,-75.893,-176.744,8.716,148.786
C09814=1149.523,321.462,-75.926,-176.742,8.720,148.786
C09815=1149.518,321.709,-75.957,-176.739,8.723,148.787
C09816=1149.514,321.957,-75.991,-176.736,8.727,148.787
C09817=1149.511,322.205,-76.022,-176.734,8.730,148.787
C09818=1149.506,322.453,-76.056,-176.732,8.734,148.787
C09819=1149.503,322.701,-76.087,-176.729,8.738,148.788
C09820=1149.498,322.949,-76.120,-176.726,8.741,148.788
C09821=1149.494,323.196,-76.153,-176.724,8.744,148.788
C09822=1149.490,323.444,-76.184,-176.721,8.748,148.788
C09823=1149.486,323.692,-76.218,-176.719,8.752,148.788
C09824=1149.482,323.940,-76.249,-176.716,8.756,148.789
C09825=1149.478,324.188,-76.283,-176.714,8.759,148.789
C09826=1149.473,324.436,-76.315,-176.711,8.762,148.789
C09827=1149.470,324.683,-76.348,-176.708,8.766,148.789
C09828=1149.466,324.932,-76.380,-176.706,8.769,148.789
C09829=1149.461,325.179,-76.413,-176.703,8.773,148.789
C09830=1149.457,325.427,-76.445,-176.700,8.777,148.790
C09831=1149.453,325.674,-76.478,-176.698,8.780,148.790
C09832=1149.449,325.923,-76.510,-176.695,8.784,148.790
C09833=1149.445,326.170,-76.543,-176.693,8.787,148.790
C09834=1149.441,326.418,-76.576,-176.691,8.791,148.790
C09835=1149.437,326.666,-76.608,-176.688,8.795,148.791
C09836=1149.433,326.914,-76.641,-176.685,8.798,148.791
C09837=1149.429,327.162,-76.673,-176.682,8.802,148.791
C09838=1149.425,327.410,-76.707,-176.680,8.805,148.791
C09839=1149.420,327.658,-76.740,-176.678,8.809,148.791
C09840=1149.417,327.905,-76.772,-176.675,8.813,148.792
C09841=1149.413,328.153,-76.805,-176.673,8.816,148.792
C09842=1149.408,328.401,-76.838,-176.670,8.820,148.792
C09843=1149.404,328.649,-76.871,-176.667,8.823,148.792
C09844=1149.401,328.897,-76.903,-176.664,8.827,148.793
C09845=1149.396,329.145,-76.936,-176.662,8.831,148.793
C09846=1149.392,329.392,-76.969,-176.660,8.834,148.793
C09847=1149.388,329.640,-77.002,-176.657,8.838,148.793
C09848=1149.384,329.888,-77.036,-176.655,8.841,148.793
C09849=1149.380,330.136,-77.068,-176.652,8.845,148.794
C09850=1149.376,330.383,-77.101,-176.649,8.849,148.794
C09851=1149.372,330.631,-77.134,-176.647,8.852,148.794
C09852=1149.368,330.879,-77.167,-176.644,8.856,148.794
C09853=1149.364,331.127,-77.200,-176.642,8.859,148.794
C09854=1149.360,331.374,-77.233,-176.639,8.864,148.795
C09855=1149.356,331.622,-77.266,-176.637,8.867,148.795
C09856=1149.351,331.870,-77.299,-176.634,8.871,148.795
C09857=1149.347,332.118,-77.333,-176.632,8.874,148.796
C09858=1149.343,332.366,-77.365,-176.629,8.878,148.796
C09859=1149.339,332.613,-77.398,-176.626,8.882,148.796
C09860=1149.335,332.861,-77.431,-176.624,8.885,148.796
C09861=1149.331,333.109,-77.464,-176.621,8.889,148.796
C09862=1149.327,333.357,-77.497,-176.619,8.892,148.797
C09863=1149.323,333.604,-77.530,-176.616,8.896,148.797
C09864=1149.319,333.852,-77.563,-176.614,8.900,148.797
C09865=1149.315,334.099,-77.597,-176.611,8.904,148.797
C09866=1149.311,334.347,-77.630,-176.608,8.907,148.798
C09867=1149.307,334.595,-77.664,-176.607,8.911,148.798
C09868=1149.303,334.843,-77.697,-176.604,8.915,148.798
C09869=1149.299,335.091,-77.730,-176.601,8.918,148.798
C09870=1149.295,335.338,-77.763,-176.598,8.922,148.799
C09871=1149.291,335.586,-77.797,-176.596,8.925,148.799
C09872=1149.287,335.834,-77.830,-176.593,8.929,148.799
C09873=1149.283,336.081,-77.864,-176.591,8.933,148.799
C09874=1149.279,336.329,-77.897,-176.588,8.937,148.799
C09875=1149.275,336.577,-77.930,-176.586,8.940,148.800
C09876=1149.270,336.825,-77.964,-176.583,8.944,148.800
C09877=1149.266,337.073,-77.997,-176.581,8.948,148.800
C09878=1149.262,337.320,-78.031,-176.578,8.952,148.801
C09879=1149.258,337.568,-78.064,-176.576,8.955,148.801
C09880=1149.254,337.815,-78.097,-176.573,8.958,148.801
C09881=1149.250,338.064,-78.131,-176.570,8.962,148.801
C09882=1149.247,338.311,-78.165,-176.568,8.966,148.801
C09883=1149.242,338.559,-78.198,-176.566,8.970,148.802
C09884=1149.238,338.807,-78.232,-176.563,8.973,148.802
C09885=1149.234,339.087,-78.270,-176.560,8.978,148.802
C09886=1149.229,339.367,-78.307,-176.557,8.982,148.803
C09887=1149.224,339.647,-78.346,-176.554,8.987,148.803
C09888=1149.220,339.928,-78.383,-176.552,8.991,148.803
C09889=1149.216,340.175,-78.418,-176.549,8.994,148.804
C09890=1149.211,340.423,-78.451,-176.546,8.998,148.804
C09891=1149.207,340.670,-78.484,-176.544,9.002,148.804
C09892=1149.204,340.918,-78.519,-176.541,9.006,148.804
C09893=1149.199,341.166,-78.552,-176.539,9.009,148.804
C09894=1149.195,341.413,-78.586,-176.536,9.013,148.805
C09895=1149.191,341.661,-78.619,-176.534,9.017,148.805
C09896=1149.188,341.909,-78.654,-176.531,9.021,148.805
C09897=1149.183,342.157,-78.687,-176.529,9.024,148.806
C09898=1149.179,342.404,-78.721,-176.526,9.028,148.806
C09899=1149.175,342.652,-78.754,-176.524,9.032,148.806
C09900=1149.171,342.900,-78.789,-176.521,9.036,148.806
C09901=1149.167,343.147,-78.823,-176.519,9.039,148.807
C09902=1149.163,343.395,-78.856,-176.516,9.043,148.807
C09903=1149.159,343.642,-78.891,-176.514,9.047,148.807
C09904=1149.155,343.891,-78.924,-176.511,9.051,148.808
C09905=1149.151,344.138,-78.958,-176.509,9.054,148.808
C09906=1149.147,344.385,-78.992,-176.506,9.058,148.808
C09907=1149.143,344.634,-79.026,-176.504,9.062,148.808
C09908=1149.139,344.881,-79.060,-176.501,9.066,148.809
C09909=1149.135,345.128,-79.094,-176.499,9.069,148.809
C09910=1149.131,345.377,-79.128,-176.496,9.073,148.809
C09911=1149.127,345.624,-79.162,-176.494,9.077,148.809
C09912=1149.123,345.871,-79.196,-176.491,9.081,148.810
C09913=1149.119,346.119,-79.231,-176.489,9.084,148.810
C09914=1149.115,346.366,-79.265,-176.486,9.088,148.810
C09915=1149.111,346.614,-79.298,-176.483,9.093,148.811
C09916=1149.107,346.862,-79.333,-176.481,9.096,148.811
C09917=1149.103,347.109,-79.367,-176.478,9.100,148.811
C09918=1149.099,347.357,-79.402,-176.476,9.103,148.812
C09919=1149.095,347.605,-79.435,-176.473,9.108,148.812
C09920=1149.090,347.853,-79.469,-176.471,9.111,148.812
C09921=1149.087,348.100,-79.503,-176.468,9.115,148.812
C09922=1149.083,348.348,-79.538,-176.466,9.119,148.813
C09923=1149.079,348.596,-79.572,-176.463,9.123,148.813
C09924=1149.075,348.843,-79.607,-176.461,9.126,148.813
C09925=1149.071,349.090,-79.641,-176.458,9.130,148.814
C09926=1149.067,349.338,-79.675,-176.455,9.134,148.814
C09927=1149.063,349.585,-79.709,-176.453,9.138,148.814
C09928=1149.059,349.833,-79.744,-176.451,9.142,148.814
C09929=1149.055,350.081,-79.779,-176.448,9.145,148.815
C09930=1149.051,350.329,-79.813,-176.445,9.149,148.815
C09931=1149.047,350.576,-79.847,-176.443,9.153,148.815
C09932=1149.043,350.823,-79.881,-176.441,9.157,148.816
C09933=1149.039,351.071,-79.916,-176.438,9.160,148.816
C09934=1149.035,351.319,-79.950,-176.436,9.165,148.816
C09935=1149.031,351.567,-79.985,-176.433,9.169,148.817
C09936=1149.027,351.814,-80.019,-176.430,9.172,148.817
C09937=1149.023,352.062,-80.053,-176.428,9.176,148.817
C09938=1149.019,352.309,-80.089,-176.426,9.180,148.817
C09939=1149.015,352.557,-80.123,-176.423,9.184,148.818
C09940=1149.011,352.804,-80.157,-176.420,9.188,148.818
C09941=1149.007,353.052,-80.192,-176.418,9.192,148.818
C09942=1149.003,353.299,-80.227,-176.415,9.196,148.819
C09943=1149.000,353.547,-80.261,-176.413,9.199,148.819
C09944=1148.995,353.794,-80.296,-176.410,9.203,148.819
C09945=1148.991,354.042,-80.331,-176.408,9.207,148.819
C09946=1148.987,354.290,-80.365,-176.405,9.211,148.820
C09947=1148.984,354.537,-80.399,-176.403,9.215,148.820
C09948=1148.980,354.785,-80.435,-176.401,9.219,148.821
C09949=1148.975,355.032,-80.469,-176.398,9.223,148.821
C09950=1148.972,355.280,-80.504,-176.395,9.226,148.821
C09951=1148.968,355.527,-80.539,-176.393,9.230,148.822
C09952=1148.964,355.775,-80.574,-176.390,9.234,148.822
C09953=1148.959,356.022,-80.608,-176.388,9.238,148.822
C09954=1148.956,356.270,-80.644,-176.385,9.242,148.822
C09955=1148.952,356.518,-80.678,-176.383,9.245,148.823
C09956=1148.948,356.765,-80.712,-176.380,9.250,148.823
C09957=1148.944,357.013,-80.748,-176.377,9.254,148.823
C09958=1148.940,357.260,-80.782,-176.376,9.257,148.824
C09959=1148.936,357.508,-80.818,-176.373,9.262,148.824
C09960=1148.933,357.755,-80.852,-176.370,9.266,148.824
C09961=1148.928,358.002,-80.887,-176.368,9.269,148.825
C09962=1148.925,358.250,-80.922,-176.365,9.273,148.825
C09963=1148.921,358.498,-80.958,-176.363,9.277,148.825
C09964=1148.916,358.745,-80.992,-176.360,9.281,148.826
C09965=1148.913,358.993,-81.028,-176.357,9.285,148.826
C09966=1148.908,359.240,-81.062,-176.355,9.289,148.826
C09967=1148.904,359.488,-81.098,-176.352,9.293,148.827
C09968=1148.901,359.735,-81.132,-176.350,9.297,148.827
C09969=1148.897,359.983,-81.168,-176.348,9.300,148.827
C09970=1148.893,360.230,-81.203,-176.345,9.304,148.828
C09971=1148.889,360.478,-81.238,-176.342,9.309,148.828
C09972=1148.886,360.725,-81.273,-176.340,9.312,148.828
C09973=1148.881,360.973,-81.308,-176.337,9.317,148.829
C09974=1148.877,361.220,-81.343,-176.334,9.321,148.829
C09975=1148.874,361.468,-81.379,-176.332,9.325,148.829
C09976=1148.869,361.715,-81.414,-176.330,9.328,148.830
C09977=1148.865,361.963,-81.449,-176.327,9.332,148.830
C09978=1148.862,362.210,-81.484,-176.324,9.337,148.830
C09979=1148.858,362.458,-81.520,-176.321,9.341,148.831
C09980=1148.854,362.705,-81.554,-176.319,9.344,148.831
C09981=1148.850,362.953,-81.590,-176.317,9.349,148.831
C09982=1148.846,363.200,-81.625,-176.314,9.353,148.832
C09983=1148.843,363.448,-81.661,-176.311,9.357,148.832
C09984=1148.838,363.694,-81.696,-176.309,9.360,148.832
C09985=1148.835,363.942,-81.732,-176.306,9.365,148.833
C09986=1148.831,364.190,-81.767,-176.303,9.369,148.833
C09987=1148.827,364.438,-81.802,-176.301,9.373,148.833
C09988=1148.823,364.684,-81.837,-176.299,9.376,148.834
C09989=1148.818,364.968,-81.878,-176.296,9.382,148.834
C09990=1148.814,365.251,-81.919,-176.293,9.386,148.834
C09991=1148.810,365.534,-81.960,-176.290,9.391,148.835
C09992=1148.805,365.818,-82.000,-176.287,9.395,148.835
C09993=1148.801,366.065,-82.036,-176.284,9.399,148.836
C09994=1148.797,366.312,-82.071,-176.281,9.404,148.836
C09995=1148.793,366.560,-82.107,-176.279,9.408,148.836
C09996=1148.789,366.807,-82.143,-176.276,9.411,148.837
//INST
///DATE 2021/06/15 17:26
///ATTR SC,RW,RJ
////FRAME ROBOT
///GROUP1 RB1
NOP
MOVL C00000 V=800.0 PL=0
MOVL C00001 V=800.0 PL=0
MOVL C00002 V=800.0 PL=0
MOVL C00003 V=800.0 PL=0
MOVL C00004 V=800.0 PL=0
MOVL C00005 V=800.0 PL=0
MOVL C00006 V=800.0 PL=0
MOVL C00007 V=800.0 PL=0
MOVL C00008 V=800.0 PL=0
MOVL C00009 V=800.0 PL=0
MOVL C00010 V=800.0 PL=0
MOVL C00011 V=800.0 PL=0
MOVL C00012 V=800.0 PL=0
MOVL C00013 V=800.0 PL=0
MOVL C00014 V=800.0 PL=0
MOVL C00015 V=800.0 PL=0
MOVL C00016 V=800.0 PL=0
MOVL C00017 V=800.0 PL=0
MOVL C00018 V=800.0 PL=0
MOVL C00019 V=800.0 PL=0
MOVL C00020 V=800.0 PL=0
MOVL C00021 V=800.0 PL=0
MOVL C00022 V=800.0 PL=0
MOVL C00023 V=800.0 PL=0
MOVL C00024 V=800.0 PL=0
MOVL C00025 V=800.0 PL=0
MOVL C00026 V=800.0 PL=0
MOVL C00027 V=800.0 PL=0
MOVL C00028 V=800.0 PL=0
MOVL C00029 V=800.0 PL=0
MOVL C00030 V=800.0 PL=0
MOVL C00031 V=800.0 PL=0
MOVL C00032 V=800.0 PL=0
MOVL C00033 V=800.0 PL=0
MOVL C00034 V=800.0 PL=0
MOVL C00035 V=800.0 PL=0
MOVL C00036 V=800.0 PL=0
MOVL C00037 V=800.0 PL=0
MOVL C00038 V=800.0 PL=0
MOVL C00039 V=800.0 PL=0
MOVL C00040 V=800.0 PL=0
MOVL C00041 V=800.0 PL=0
MOVL C00042 V=800.0 PL=0
MOVL C00043 V=800.0 PL=0
MOVL C00044 V=800.0 PL=0
MOVL C00045 V=800.0 PL=0
MOVL C00046 V=800.0 PL=0
MOVL C00047 V=800.0 PL=0
MOVL C00048 V=800.0 PL=0
MOVL C00049 V=800.0 PL=0
MOVL C00050 V=800.0 PL=0
MOVL C00051 V=800.0 PL=0
MOVL C00052 V=800.0 PL=0
MOVL C00053 V=800.0 PL=0
MOVL C00054 V=800.0 PL=0
MOVL C00055 V=800.0 PL=0
MOVL C00056 V=800.0 PL=0
MOVL C00057 V=800.0 PL=0
MOVL C00058 V=800.0 PL=0
MOVL C00059 V=800.0 PL=0
MOVL C00060 V=800.0 PL=0
MOVL C00061 V=800.0 PL=0
MOVL C00062 V=800.0 PL=0
MOVL C00063 V=800.0 PL=0
MOVL C00064 V=800.0 PL=0
MOVL C00065 V=800.0 PL=0
MOVL C00066 V=800.0 PL=0
MOVL C00067 V=800.0 PL=0
MOVL C00068 V=800.0 PL=0
MOVL C00069 V=800.0 PL=0
MOVL C00070 V=800.0 PL=0
MOVL C00071 V=800.0 PL=0
MOVL C00072 V=800.0 PL=0
MOVL C00073 V=800.0 PL=0
MOVL C00074 V=800.0 PL=0
MOVL C00075 V=800.0 PL=0
MOVL C00076 V=800.0 PL=0
MOVL C00077 V=800.0 PL=0
MOVL C00078 V=800.0 PL=0
MOVL C00079 V=800.0 PL=0
MOVL C00080 V=800.0 PL=0
MOVL C00081 V=800.0 PL=0
MOVL C00082 V=800.0 PL=0
MOVL C00083 V=800.0 PL=0
MOVL C00084 V=800.0 PL=0
MOVL C00085 V=800.0 PL=0
MOVL C00086 V=800.0 PL=0
MOVL C00087 V=800.0 PL=0
MOVL C00088 V=800.0 PL=0
MOVL C00089 V=800.0 PL=0
MOVL C00090 V=800.0 PL=0
MOVL C00091 V=800.0 PL=0
MOVL C00092 V=800.0 PL=0
MOVL C00093 V=800.0 PL=0
MOVL C00094 V=800.0 PL=0
MOVL C00095 V=800.0 PL=0
MOVL C00096 V=800.0 PL=0
MOVL C00097 V=800.0 PL=0
MOVL C00098 V=800.0 PL=0
MOVL C00099 V=800.0 PL=0
MOVL C00100 V=800.0 PL=0
MOVL C00101 V=800.0 PL=0
MOVL C00102 V=800.0 PL=0
MOVL C00103 V=800.0 PL=0
MOVL C00104 V=800.0 PL=0
MOVL C00105 V=800.0 PL=0
MOVL C00106 V=800.0 PL=0
MOVL C00107 V=800.0 PL=0
MOVL C00108 V=800.0 PL=0
MOVL C00109 V=800.0 PL=0
MOVL C00110 V=800.0 PL=0
MOVL C00111 V=800.0 PL=0
MOVL C00112 V=800.0 PL=0
MOVL C00113 V=800.0 PL=0
MOVL C00114 V=800.0 PL=0
MOVL C00115 V=800.0 PL=0
MOVL C00116 V=800.0 PL=0
MOVL C00117 V=800.0 PL=0
MOVL C00118 V=800.0 PL=0
MOVL C00119 V=800.0 PL=0
MOVL C00120 V=800.0 PL=0
MOVL C00121 V=800.0 PL=0
MOVL C00122 V=800.0 PL=0
MOVL C00123 V=800.0 PL=0
MOVL C00124 V=800.0 PL=0
MOVL C00125 V=800.0 PL=0
MOVL C00126 V=800.0 PL=0
MOVL C00127 V=800.0 PL=0
MOVL C00128 V=800.0 PL=0
MOVL C00129 V=800.0 PL=0
MOVL C00130 V=800.0 PL=0
MOVL C00131 V=800.0 PL=0
MOVL C00132 V=800.0 PL=0
MOVL C00133 V=800.0 PL=0
MOVL C00134 V=800.0 PL=0
MOVL C00135 V=800.0 PL=0
MOVL C00136 V=800.0 PL=0
MOVL C00137 V=800.0 PL=0
MOVL C00138 V=800.0 PL=0
MOVL C00139 V=800.0 PL=0
MOVL C00140 V=800.0 PL=0
MOVL C00141 V=800.0 PL=0
MOVL C00142 V=800.0 PL=0
MOVL C00143 V=800.0 PL=0
MOVL C00144 V=800.0 PL=0
MOVL C00145 V=800.0 PL=0
MOVL C00146 V=800.0 PL=0
MOVL C00147 V=800.0 PL=0
MOVL C00148 V=800.0 PL=0
MOVL C00149 V=800.0 PL=0
MOVL C00150 V=800.0 PL=0
MOVL C00151 V=800.0 PL=0
MOVL C00152 V=800.0 PL=0
MOVL C00153 V=800.0 PL=0
MOVL C00154 V=800.0 PL=0
MOVL C00155 V=800.0 PL=0
MOVL C00156 V=800.0 PL=0
MOVL C00157 V=800.0 PL=0
MOVL C00158 V=800.0 PL=0
MOVL C00159 V=800.0 PL=0
MOVL C00160 V=800.0 PL=0
MOVL C00161 V=800.0 PL=0
MOVL C00162 V=800.0 PL=0
MOVL C00163 V=800.0 PL=0
MOVL C00164 V=800.0 PL=0
MOVL C00165 V=800.0 PL=0
MOVL C00166 V=800.0 PL=0
MOVL C00167 V=800.0 PL=0
MOVL C00168 V=800.0 PL=0
MOVL C00169 V=800.0 PL=0
MOVL C00170 V=800.0 PL=0
MOVL C00171 V=800.0 PL=0
MOVL C00172 V=800.0 PL=0
MOVL C00173 V=800.0 PL=0
MOVL C00174 V=800.0 PL=0
MOVL C00175 V=800.0 PL=0
MOVL C00176 V=800.0 PL=0
MOVL C00177 V=800.0 PL=0
MOVL C00178 V=800.0 PL=0
MOVL C00179 V=800.0 PL=0
MOVL C00180 V=800.0 PL=0
MOVL C00181 V=800.0 PL=0
MOVL C00182 V=800.0 PL=0
MOVL C00183 V=800.0 PL=0
MOVL C00184 V=800.0 PL=0
MOVL C00185 V=800.0 PL=0
MOVL C00186 V=800.0 PL=0
MOVL C00187 V=800.0 PL=0
MOVL C00188 V=800.0 PL=0
MOVL C00189 V=800.0 PL=0
MOVL C00190 V=800.0 PL=0
MOVL C00191 V=800.0 PL=0
MOVL C00192 V=800.0 PL=0
MOVL C00193 V=800.0 PL=0
MOVL C00194 V=800.0 PL=0
MOVL C00195 V=800.0 PL=0
MOVL C00196 V=800.0 PL=0
MOVL C00197 V=800.0 PL=0
MOVL C00198 V=800.0 PL=0
MOVL C00199 V=800.0 PL=0
MOVL C00200 V=800.0 PL=0
MOVL C00201 V=800.0 PL=0
MOVL C00202 V=800.0 PL=0
MOVL C00203 V=800.0 PL=0
MOVL C00204 V=800.0 PL=0
MOVL C00205 V=800.0 PL=0
MOVL C00206 V=800.0 PL=0
MOVL C00207 V=800.0 PL=0
MOVL C00208 V=800.0 PL=0
MOVL C00209 V=800.0 PL=0
MOVL C00210 V=800.0 PL=0
MOVL C00211 V=800.0 PL=0
MOVL C00212 V=800.0 PL=0
MOVL C00213 V=800.0 PL=0
MOVL C00214 V=800.0 PL=0
MOVL C00215 V=800.0 PL=0
MOVL C00216 V=800.0 PL=0
MOVL C00217 V=800.0 PL=0
MOVL C00218 V=800.0 PL=0
MOVL C00219 V=800.0 PL=0
MOVL C00220 V=800.0 PL=0
MOVL C00221 V=800.0 PL=0
MOVL C00222 V=800.0 PL=0
MOVL C00223 V=800.0 PL=0
MOVL C00224 V=800.0 PL=0
MOVL C00225 V=800.0 PL=0
MOVL C00226 V=800.0 PL=0
MOVL C00227 V=800.0 PL=0
MOVL C00228 V=800.0 PL=0
MOVL C00229 V=800.0 PL=0
MOVL C00230 V=800.0 PL=0
MOVL C00231 V=800.0 PL=0
MOVL C00232 V=800.0 PL=0
MOVL C00233 V=800.0 PL=0
MOVL C00234 V=800.0 PL=0
MOVL C00235 V=800.0 PL=0
MOVL C00236 V=800.0 PL=0
MOVL C00237 V=800.0 PL=0
MOVL C00238 V=800.0 PL=0
MOVL C00239 V=800.0 PL=0
MOVL C00240 V=800.0 PL=0
MOVL C00241 V=800.0 PL=0
MOVL C00242 V=800.0 PL=0
MOVL C00243 V=800.0 PL=0
MOVL C00244 V=800.0 PL=0
MOVL C00245 V=800.0 PL=0
MOVL C00246 V=800.0 PL=0
MOVL C00247 V=800.0 PL=0
MOVL C00248 V=800.0 PL=0
MOVL C00249 V=800.0 PL=0
MOVL C00250 V=800.0 PL=0
MOVL C00251 V=800.0 PL=0
MOVL C00252 V=800.0 PL=0
MOVL C00253 V=800.0 PL=0
MOVL C00254 V=800.0 PL=0
MOVL C00255 V=800.0 PL=0
MOVL C00256 V=800.0 PL=0
MOVL C00257 V=800.0 PL=0
MOVL C00258 V=800.0 PL=0
MOVL C00259 V=800.0 PL=0
MOVL C00260 V=800.0 PL=0
MOVL C00261 V=800.0 PL=0
MOVL C00262 V=800.0 PL=0
MOVL C00263 V=800.0 PL=0
MOVL C00264 V=800.0 PL=0
MOVL C00265 V=800.0 PL=0
MOVL C00266 V=800.0 PL=0
MOVL C00267 V=800.0 PL=0
MOVL C00268 V=800.0 PL=0
MOVL C00269 V=800.0 PL=0
MOVL C00270 V=800.0 PL=0
MOVL C00271 V=800.0 PL=0
MOVL C00272 V=800.0 PL=0
MOVL C00273 V=800.0 PL=0
MOVL C00274 V=800.0 PL=0
MOVL C00275 V=800.0 PL=0
MOVL C00276 V=800.0 PL=0
MOVL C00277 V=800.0 PL=0
MOVL C00278 V=800.0 PL=0
MOVL C00279 V=800.0 PL=0
MOVL C00280 V=800.0 PL=0
MOVL C00281 V=800.0 PL=0
MOVL C00282 V=800.0 PL=0
MOVL C00283 V=800.0 PL=0
MOVL C00284 V=800.0 PL=0
MOVL C00285 V=800.0 PL=0
MOVL C00286 V=800.0 PL=0
MOVL C00287 V=800.0 PL=0
MOVL C00288 V=800.0 PL=0
MOVL C00289 V=800.0 PL=0
MOVL C00290 V=800.0 PL=0
MOVL C00291 V=800.0 PL=0
MOVL C00292 V=800.0 PL=0
MOVL C00293 V=800.0 PL=0
MOVL C00294 V=800.0 PL=0
MOVL C00295 V=800.0 PL=0
MOVL C00296 V=800.0 PL=0
MOVL C00297 V=800.0 PL=0
MOVL C00298 V=800.0 PL=0
MOVL C00299 V=800.0 PL=0
MOVL C00300 V=800.0 PL=0
MOVL C00301 V=800.0 PL=0
MOVL C00302 V=800.0 PL=0
MOVL C00303 V=800.0 PL=0
MOVL C00304 V=800.0 PL=0
MOVL C00305 V=800.0 PL=0
MOVL C00306 V=800.0 PL=0
MOVL C00307 V=800.0 PL=0
MOVL C00308 V=800.0 PL=0
MOVL C00309 V=800.0 PL=0
MOVL C00310 V=800.0 PL=0
MOVL C00311 V=800.0 PL=0
MOVL C00312 V=800.0 PL=0
MOVL C00313 V=800.0 PL=0
MOVL C00314 V=800.0 PL=0
MOVL C00315 V=800.0 PL=0
MOVL C00316 V=800.0 PL=0
MOVL C00317 V=800.0 PL=0
MOVL C00318 V=800.0 PL=0
MOVL C00319 V=800.0 PL=0
MOVL C00320 V=800.0 PL=0
MOVL C00321 V=800.0 PL=0
MOVL C00322 V=800.0 PL=0
MOVL C00323 V=800.0 PL=0
MOVL C00324 V=800.0 PL=0
MOVL C00325 V=800.0 PL=0
MOVL C00326 V=800.0 PL=0
MOVL C00327 V=800.0 PL=0
MOVL C00328 V=800.0 PL=0
MOVL C00329 V=800.0 PL=0
MOVL C00330 V=800.0 PL=0
MOVL C00331 V=800.0 PL=0
MOVL C00332 V=800.0 PL=0
MOVL C00333 V=800.0 PL=0
MOVL C00334 V=800.0 PL=0
MOVL C00335 V=800.0 PL=0
MOVL C00336 V=800.0 PL=0
MOVL C00337 V=800.0 PL=0
MOVL C00338 V=800.0 PL=0
MOVL C00339 V=800.0 PL=0
MOVL C00340 V=800.0 PL=0
MOVL C00341 V=800.0 PL=0
MOVL C00342 V=800.0 PL=0
MOVL C00343 V=800.0 PL=0
MOVL C00344 V=800.0 PL=0
MOVL C00345 V=800.0 PL=0
MOVL C00346 V=800.0 PL=0
MOVL C00347 V=800.0 PL=0
MOVL C00348 V=800.0 PL=0
MOVL C00349 V=800.0 PL=0
MOVL C00350 V=800.0 PL=0
MOVL C00351 V=800.0 PL=0
MOVL C00352 V=800.0 PL=0
MOVL C00353 V=800.0 PL=0
MOVL C00354 V=800.0 PL=0
MOVL C00355 V=800.0 PL=0
MOVL C00356 V=800.0 PL=0
MOVL C00357 V=800.0 PL=0
MOVL C00358 V=800.0 PL=0
MOVL C00359 V=800.0 PL=0
MOVL C00360 V=800.0 PL=0
MOVL C00361 V=800.0 PL=0
MOVL C00362 V=800.0 PL=0
MOVL C00363 V=800.0 PL=0
MOVL C00364 V=800.0 PL=0
MOVL C00365 V=800.0 PL=0
MOVL C00366 V=800.0 PL=0
MOVL C00367 V=800.0 PL=0
MOVL C00368 V=800.0 PL=0
MOVL C00369 V=800.0 PL=0
MOVL C00370 V=800.0 PL=0
MOVL C00371 V=800.0 PL=0
MOVL C00372 V=800.0 PL=0
MOVL C00373 V=800.0 PL=0
MOVL C00374 V=800.0 PL=0
MOVL C00375 V=800.0 PL=0
MOVL C00376 V=800.0 PL=0
MOVL C00377 V=800.0 PL=0
MOVL C00378 V=800.0 PL=0
MOVL C00379 V=800.0 PL=0
MOVL C00380 V=800.0 PL=0
MOVL C00381 V=800.0 PL=0
MOVL C00382 V=800.0 PL=0
MOVL C00383 V=800.0 PL=0
MOVL C00384 V=800.0 PL=0
MOVL C00385 V=800.0 PL=0
MOVL C00386 V=800.0 PL=0
MOVL C00387 V=800.0 PL=0
MOVL C00388 V=800.0 PL=0
MOVL C00389 V=800.0 PL=0
MOVL C00390 V=800.0 PL=0
MOVL C00391 V=800.0 PL=0
MOVL C00392 V=800.0 PL=0
MOVL C00393 V=800.0 PL=0
MOVL C00394 V=800.0 PL=0
MOVL C00395 V=800.0 PL=0
MOVL C00396 V=800.0 PL=0
MOVL C00397 V=800.0 PL=0
MOVL C00398 V=800.0 PL=0
MOVL C00399 V=800.0 PL=0
MOVL C00400 V=800.0 PL=0
MOVL C00401 V=800.0 PL=0
MOVL C00402 V=800.0 PL=0
MOVL C00403 V=800.0 PL=0
MOVL C00404 V=800.0 PL=0
MOVL C00405 V=800.0 PL=0
MOVL C00406 V=800.0 PL=0
MOVL C00407 V=800.0 PL=0
MOVL C00408 V=800.0 PL=0
MOVL C00409 V=800.0 PL=0
MOVL C00410 V=800.0 PL=0
MOVL C00411 V=800.0 PL=0
MOVL C00412 V=800.0 PL=0
MOVL C00413 V=800.0 PL=0
MOVL C00414 V=800.0 PL=0
MOVL C00415 V=800.0 PL=0
MOVL C00416 V=800.0 PL=0
MOVL C00417 V=800.0 PL=0
MOVL C00418 V=800.0 PL=0
MOVL C00419 V=800.0 PL=0
MOVL C00420 V=800.0 PL=0
MOVL C00421 V=800.0 PL=0
MOVL C00422 V=800.0 PL=0
MOVL C00423 V=800.0 PL=0
MOVL C00424 V=800.0 PL=0
MOVL C00425 V=800.0 PL=0
MOVL C00426 V=800.0 PL=0
MOVL C00427 V=800.0 PL=0
MOVL C00428 V=800.0 PL=0
MOVL C00429 V=800.0 PL=0
MOVL C00430 V=800.0 PL=0
MOVL C00431 V=800.0 PL=0
MOVL C00432 V=800.0 PL=0
MOVL C00433 V=800.0 PL=0
MOVL C00434 V=800.0 PL=0
MOVL C00435 V=800.0 PL=0
MOVL C00436 V=800.0 PL=0
MOVL C00437 V=800.0 PL=0
MOVL C00438 V=800.0 PL=0
MOVL C00439 V=800.0 PL=0
MOVL C00440 V=800.0 PL=0
MOVL C00441 V=800.0 PL=0
MOVL C00442 V=800.0 PL=0
MOVL C00443 V=800.0 PL=0
MOVL C00444 V=800.0 PL=0
MOVL C00445 V=800.0 PL=0
MOVL C00446 V=800.0 PL=0
MOVL C00447 V=800.0 PL=0
MOVL C00448 V=800.0 PL=0
MOVL C00449 V=800.0 PL=0
MOVL C00450 V=800.0 PL=0
MOVL C00451 V=800.0 PL=0
MOVL C00452 V=800.0 PL=0
MOVL C00453 V=800.0 PL=0
MOVL C00454 V=800.0 PL=0
MOVL C00455 V=800.0 PL=0
MOVL C00456 V=800.0 PL=0
MOVL C00457 V=800.0 PL=0
MOVL C00458 V=800.0 PL=0
MOVL C00459 V=800.0 PL=0
MOVL C00460 V=800.0 PL=0
MOVL C00461 V=800.0 PL=0
MOVL C00462 V=800.0 PL=0
MOVL C00463 V=800.0 PL=0
MOVL C00464 V=800.0 PL=0
MOVL C00465 V=800.0 PL=0
MOVL C00466 V=800.0 PL=0
MOVL C00467 V=800.0 PL=0
MOVL C00468 V=800.0 PL=0
MOVL C00469 V=800.0 PL=0
MOVL C00470 V=800.0 PL=0
MOVL C00471 V=800.0 PL=0
MOVL C00472 V=800.0 PL=0
MOVL C00473 V=800.0 PL=0
MOVL C00474 V=800.0 PL=0
MOVL C00475 V=800.0 PL=0
MOVL C00476 V=800.0 PL=0
MOVL C00477 V=800.0 PL=0
MOVL C00478 V=800.0 PL=0
MOVL C00479 V=800.0 PL=0
MOVL C00480 V=800.0 PL=0
MOVL C00481 V=800.0 PL=0
MOVL C00482 V=800.0 PL=0
MOVL C00483 V=800.0 PL=0
MOVL C00484 V=800.0 PL=0
MOVL C00485 V=800.0 PL=0
MOVL C00486 V=800.0 PL=0
MOVL C00487 V=800.0 PL=0
MOVL C00488 V=800.0 PL=0
MOVL C00489 V=800.0 PL=0
MOVL C00490 V=800.0 PL=0
MOVL C00491 V=800.0 PL=0
MOVL C00492 V=800.0 PL=0
MOVL C00493 V=800.0 PL=0
MOVL C00494 V=800.0 PL=0
MOVL C00495 V=800.0 PL=0
MOVL C00496 V=800.0 PL=0
MOVL C00497 V=800.0 PL=0
MOVL C00498 V=800.0 PL=0
MOVL C00499 V=800.0 PL=0
MOVL C00500 V=800.0 PL=0
MOVL C00501 V=800.0 PL=0
MOVL C00502 V=800.0 PL=0
MOVL C00503 V=800.0 PL=0
MOVL C00504 V=800.0 PL=0
MOVL C00505 V=800.0 PL=0
MOVL C00506 V=800.0 PL=0
MOVL C00507 V=800.0 PL=0
MOVL C00508 V=800.0 PL=0
MOVL C00509 V=800.0 PL=0
MOVL C00510 V=800.0 PL=0
MOVL C00511 V=800.0 PL=0
MOVL C00512 V=800.0 PL=0
MOVL C00513 V=800.0 PL=0
MOVL C00514 V=800.0 PL=0
MOVL C00515 V=800.0 PL=0
MOVL C00516 V=800.0 PL=0
MOVL C00517 V=800.0 PL=0
MOVL C00518 V=800.0 PL=0
MOVL C00519 V=800.0 PL=0
MOVL C00520 V=800.0 PL=0
MOVL C00521 V=800.0 PL=0
MOVL C00522 V=800.0 PL=0
MOVL C00523 V=800.0 PL=0
MOVL C00524 V=800.0 PL=0
MOVL C00525 V=800.0 PL=0
MOVL C00526 V=800.0 PL=0
MOVL C00527 V=800.0 PL=0
MOVL C00528 V=800.0 PL=0
MOVL C00529 V=800.0 PL=0
MOVL C00530 V=800.0 PL=0
MOVL C00531 V=800.0 PL=0
MOVL C00532 V=800.0 PL=0
MOVL C00533 V=800.0 PL=0
MOVL C00534 V=800.0 PL=0
MOVL C00535 V=800.0 PL=0
MOVL C00536 V=800.0 PL=0
MOVL C00537 V=800.0 PL=0
MOVL C00538 V=800.0 PL=0
MOVL C00539 V=800.0 PL=0
MOVL C00540 V=800.0 PL=0
MOVL C00541 V=800.0 PL=0
MOVL C00542 V=800.0 PL=0
MOVL C00543 V=800.0 PL=0
MOVL C00544 V=800.0 PL=0
MOVL C00545 V=800.0 PL=0
MOVL C00546 V=800.0 PL=0
MOVL C00547 V=800.0 PL=0
MOVL C00548 V=800.0 PL=0
MOVL C00549 V=800.0 PL=0
MOVL C00550 V=800.0 PL=0
MOVL C00551 V=800.0 PL=0
MOVL C00552 V=800.0 PL=0
MOVL C00553 V=800.0 PL=0
MOVL C00554 V=800.0 PL=0
MOVL C00555 V=800.0 PL=0
MOVL C00556 V=800.0 PL=0
MOVL C00557 V=800.0 PL=0
MOVL C00558 V=800.0 PL=0
MOVL C00559 V=800.0 PL=0
MOVL C00560 V=800.0 PL=0
MOVL C00561 V=800.0 PL=0
MOVL C00562 V=800.0 PL=0
MOVL C00563 V=800.0 PL=0
MOVL C00564 V=800.0 PL=0
MOVL C00565 V=800.0 PL=0
MOVL C00566 V=800.0 PL=0
MOVL C00567 V=800.0 PL=0
MOVL C00568 V=800.0 PL=0
MOVL C00569 V=800.0 PL=0
MOVL C00570 V=800.0 PL=0
MOVL C00571 V=800.0 PL=0
MOVL C00572 V=800.0 PL=0
MOVL C00573 V=800.0 PL=0
MOVL C00574 V=800.0 PL=0
MOVL C00575 V=800.0 PL=0
MOVL C00576 V=800.0 PL=0
MOVL C00577 V=800.0 PL=0
MOVL C00578 V=800.0 PL=0
MOVL C00579 V=800.0 PL=0
MOVL C00580 V=800.0 PL=0
MOVL C00581 V=800.0 PL=0
MOVL C00582 V=800.0 PL=0
MOVL C00583 V=800.0 PL=0
MOVL C00584 V=800.0 PL=0
MOVL C00585 V=800.0 PL=0
MOVL C00586 V=800.0 PL=0
MOVL C00587 V=800.0 PL=0
MOVL C00588 V=800.0 PL=0
MOVL C00589 V=800.0 PL=0
MOVL C00590 V=800.0 PL=0
MOVL C00591 V=800.0 PL=0
MOVL C00592 V=800.0 PL=0
MOVL C00593 V=800.0 PL=0
MOVL C00594 V=800.0 PL=0
MOVL C00595 V=800.0 PL=0
MOVL C00596 V=800.0 PL=0
MOVL C00597 V=800.0 PL=0
MOVL C00598 V=800.0 PL=0
MOVL C00599 V=800.0 PL=0
MOVL C00600 V=800.0 PL=0
MOVL C00601 V=800.0 PL=0
MOVL C00602 V=800.0 PL=0
MOVL C00603 V=800.0 PL=0
MOVL C00604 V=800.0 PL=0
MOVL C00605 V=800.0 PL=0
MOVL C00606 V=800.0 PL=0
MOVL C00607 V=800.0 PL=0
MOVL C00608 V=800.0 PL=0
MOVL C00609 V=800.0 PL=0
MOVL C00610 V=800.0 PL=0
MOVL C00611 V=800.0 PL=0
MOVL C00612 V=800.0 PL=0
MOVL C00613 V=800.0 PL=0
MOVL C00614 V=800.0 PL=0
MOVL C00615 V=800.0 PL=0
MOVL C00616 V=800.0 PL=0
MOVL C00617 V=800.0 PL=0
MOVL C00618 V=800.0 PL=0
MOVL C00619 V=800.0 PL=0
MOVL C00620 V=800.0 PL=0
MOVL C00621 V=800.0 PL=0
MOVL C00622 V=800.0 PL=0
MOVL C00623 V=800.0 PL=0
MOVL C00624 V=800.0 PL=0
MOVL C00625 V=800.0 PL=0
MOVL C00626 V=800.0 PL=0
MOVL C00627 V=800.0 PL=0
MOVL C00628 V=800.0 PL=0
MOVL C00629 V=800.0 PL=0
MOVL C00630 V=800.0 PL=0
MOVL C00631 V=800.0 PL=0
MOVL C00632 V=800.0 PL=0
MOVL C00633 V=800.0 PL=0
MOVL C00634 V=800.0 PL=0
MOVL C00635 V=800.0 PL=0
MOVL C00636 V=800.0 PL=0
MOVL C00637 V=800.0 PL=0
MOVL C00638 V=800.0 PL=0
MOVL C00639 V=800.0 PL=0
MOVL C00640 V=800.0 PL=0
MOVL C00641 V=800.0 PL=0
MOVL C00642 V=800.0 PL=0
MOVL C00643 V=800.0 PL=0
MOVL C00644 V=800.0 PL=0
MOVL C00645 V=800.0 PL=0
MOVL C00646 V=800.0 PL=0
MOVL C00647 V=800.0 PL=0
MOVL C00648 V=800.0 PL=0
MOVL C00649 V=800.0 PL=0
MOVL C00650 V=800.0 PL=0
MOVL C00651 V=800.0 PL=0
MOVL C00652 V=800.0 PL=0
MOVL C00653 V=800.0 PL=0
MOVL C00654 V=800.0 PL=0
MOVL C00655 V=800.0 PL=0
MOVL C00656 V=800.0 PL=0
MOVL C00657 V=800.0 PL=0
MOVL C00658 V=800.0 PL=0
MOVL C00659 V=800.0 PL=0
MOVL C00660 V=800.0 PL=0
MOVL C00661 V=800.0 PL=0
MOVL C00662 V=800.0 PL=0
MOVL C00663 V=800.0 PL=0
MOVL C00664 V=800.0 PL=0
MOVL C00665 V=800.0 PL=0
MOVL C00666 V=800.0 PL=0
MOVL C00667 V=800.0 PL=0
MOVL C00668 V=800.0 PL=0
MOVL C00669 V=800.0 PL=0
MOVL C00670 V=800.0 PL=0
MOVL C00671 V=800.0 PL=0
MOVL C00672 V=800.0 PL=0
MOVL C00673 V=800.0 PL=0
MOVL C00674 V=800.0 PL=0
MOVL C00675 V=800.0 PL=0
MOVL C00676 V=800.0 PL=0
MOVL C00677 V=800.0 PL=0
MOVL C00678 V=800.0 PL=0
MOVL C00679 V=800.0 PL=0
MOVL C00680 V=800.0 PL=0
MOVL C00681 V=800.0 PL=0
MOVL C00682 V=800.0 PL=0
MOVL C00683 V=800.0 PL=0
MOVL C00684 V=800.0 PL=0
MOVL C00685 V=800.0 PL=0
MOVL C00686 V=800.0 PL=0
MOVL C00687 V=800.0 PL=0
MOVL C00688 V=800.0 PL=0
MOVL C00689 V=800.0 PL=0
MOVL C00690 V=800.0 PL=0
MOVL C00691 V=800.0 PL=0
MOVL C00692 V=800.0 PL=0
MOVL C00693 V=800.0 PL=0
MOVL C00694 V=800.0 PL=0
MOVL C00695 V=800.0 PL=0
MOVL C00696 V=800.0 PL=0
MOVL C00697 V=800.0 PL=0
MOVL C00698 V=800.0 PL=0
MOVL C00699 V=800.0 PL=0
MOVL C00700 V=800.0 PL=0
MOVL C00701 V=800.0 PL=0
MOVL C00702 V=800.0 PL=0
MOVL C00703 V=800.0 PL=0
MOVL C00704 V=800.0 PL=0
MOVL C00705 V=800.0 PL=0
MOVL C00706 V=800.0 PL=0
MOVL C00707 V=800.0 PL=0
MOVL C00708 V=800.0 PL=0
MOVL C00709 V=800.0 PL=0
MOVL C00710 V=800.0 PL=0
MOVL C00711 V=800.0 PL=0
MOVL C00712 V=800.0 PL=0
MOVL C00713 V=800.0 PL=0
MOVL C00714 V=800.0 PL=0
MOVL C00715 V=800.0 PL=0
MOVL C00716 V=800.0 PL=0
MOVL C00717 V=800.0 PL=0
MOVL C00718 V=800.0 PL=0
MOVL C00719 V=800.0 PL=0
MOVL C00720 V=800.0 PL=0
MOVL C00721 V=800.0 PL=0
MOVL C00722 V=800.0 PL=0
MOVL C00723 V=800.0 PL=0
MOVL C00724 V=800.0 PL=0
MOVL C00725 V=800.0 PL=0
MOVL C00726 V=800.0 PL=0
MOVL C00727 V=800.0 PL=0
MOVL C00728 V=800.0 PL=0
MOVL C00729 V=800.0 PL=0
MOVL C00730 V=800.0 PL=0
MOVL C00731 V=800.0 PL=0
MOVL C00732 V=800.0 PL=0
MOVL C00733 V=800.0 PL=0
MOVL C00734 V=800.0 PL=0
MOVL C00735 V=800.0 PL=0
MOVL C00736 V=800.0 PL=0
MOVL C00737 V=800.0 PL=0
MOVL C00738 V=800.0 PL=0
MOVL C00739 V=800.0 PL=0
MOVL C00740 V=800.0 PL=0
MOVL C00741 V=800.0 PL=0
MOVL C00742 V=800.0 PL=0
MOVL C00743 V=800.0 PL=0
MOVL C00744 V=800.0 PL=0
MOVL C00745 V=800.0 PL=0
MOVL C00746 V=800.0 PL=0
MOVL C00747 V=800.0 PL=0
MOVL C00748 V=800.0 PL=0
MOVL C00749 V=800.0 PL=0
MOVL C00750 V=800.0 PL=0
MOVL C00751 V=800.0 PL=0
MOVL C00752 V=800.0 PL=0
MOVL C00753 V=800.0 PL=0
MOVL C00754 V=800.0 PL=0
MOVL C00755 V=800.0 PL=0
MOVL C00756 V=800.0 PL=0
MOVL C00757 V=800.0 PL=0
MOVL C00758 V=800.0 PL=0
MOVL C00759 V=800.0 PL=0
MOVL C00760 V=800.0 PL=0
MOVL C00761 V=800.0 PL=0
MOVL C00762 V=800.0 PL=0
MOVL C00763 V=800.0 PL=0
MOVL C00764 V=800.0 PL=0
MOVL C00765 V=800.0 PL=0
MOVL C00766 V=800.0 PL=0
MOVL C00767 V=800.0 PL=0
MOVL C00768 V=800.0 PL=0
MOVL C00769 V=800.0 PL=0
MOVL C00770 V=800.0 PL=0
MOVL C00771 V=800.0 PL=0
MOVL C00772 V=800.0 PL=0
MOVL C00773 V=800.0 PL=0
MOVL C00774 V=800.0 PL=0
MOVL C00775 V=800.0 PL=0
MOVL C00776 V=800.0 PL=0
MOVL C00777 V=800.0 PL=0
MOVL C00778 V=800.0 PL=0
MOVL C00779 V=800.0 PL=0
MOVL C00780 V=800.0 PL=0
MOVL C00781 V=800.0 PL=0
MOVL C00782 V=800.0 PL=0
MOVL C00783 V=800.0 PL=0
MOVL C00784 V=800.0 PL=0
MOVL C00785 V=800.0 PL=0
MOVL C00786 V=800.0 PL=0
MOVL C00787 V=800.0 PL=0
MOVL C00788 V=800.0 PL=0
MOVL C00789 V=800.0 PL=0
MOVL C00790 V=800.0 PL=0
MOVL C00791 V=800.0 PL=0
MOVL C00792 V=800.0 PL=0
MOVL C00793 V=800.0 PL=0
MOVL C00794 V=800.0 PL=0
MOVL C00795 V=800.0 PL=0
MOVL C00796 V=800.0 PL=0
MOVL C00797 V=800.0 PL=0
MOVL C00798 V=800.0 PL=0
MOVL C00799 V=800.0 PL=0
MOVL C00800 V=800.0 PL=0
MOVL C00801 V=800.0 PL=0
MOVL C00802 V=800.0 PL=0
MOVL C00803 V=800.0 PL=0
MOVL C00804 V=800.0 PL=0
MOVL C00805 V=800.0 PL=0
MOVL C00806 V=800.0 PL=0
MOVL C00807 V=800.0 PL=0
MOVL C00808 V=800.0 PL=0
MOVL C00809 V=800.0 PL=0
MOVL C00810 V=800.0 PL=0
MOVL C00811 V=800.0 PL=0
MOVL C00812 V=800.0 PL=0
MOVL C00813 V=800.0 PL=0
MOVL C00814 V=800.0 PL=0
MOVL C00815 V=800.0 PL=0
MOVL C00816 V=800.0 PL=0
MOVL C00817 V=800.0 PL=0
MOVL C00818 V=800.0 PL=0
MOVL C00819 V=800.0 PL=0
MOVL C00820 V=800.0 PL=0
MOVL C00821 V=800.0 PL=0
MOVL C00822 V=800.0 PL=0
MOVL C00823 V=800.0 PL=0
MOVL C00824 V=800.0 PL=0
MOVL C00825 V=800.0 PL=0
MOVL C00826 V=800.0 PL=0
MOVL C00827 V=800.0 PL=0
MOVL C00828 V=800.0 PL=0
MOVL C00829 V=800.0 PL=0
MOVL C00830 V=800.0 PL=0
MOVL C00831 V=800.0 PL=0
MOVL C00832 V=800.0 PL=0
MOVL C00833 V=800.0 PL=0
MOVL C00834 V=800.0 PL=0
MOVL C00835 V=800.0 PL=0
MOVL C00836 V=800.0 PL=0
MOVL C00837 V=800.0 PL=0
MOVL C00838 V=800.0 PL=0
MOVL C00839 V=800.0 PL=0
MOVL C00840 V=800.0 PL=0
MOVL C00841 V=800.0 PL=0
MOVL C00842 V=800.0 PL=0
MOVL C00843 V=800.0 PL=0
MOVL C00844 V=800.0 PL=0
MOVL C00845 V=800.0 PL=0
MOVL C00846 V=800.0 PL=0
MOVL C00847 V=800.0 PL=0
MOVL C00848 V=800.0 PL=0
MOVL C00849 V=800.0 PL=0
MOVL C00850 V=800.0 PL=0
MOVL C00851 V=800.0 PL=0
MOVL C00852 V=800.0 PL=0
MOVL C00853 V=800.0 PL=0
MOVL C00854 V=800.0 PL=0
MOVL C00855 V=800.0 PL=0
MOVL C00856 V=800.0 PL=0
MOVL C00857 V=800.0 PL=0
MOVL C00858 V=800.0 PL=0
MOVL C00859 V=800.0 PL=0
MOVL C00860 V=800.0 PL=0
MOVL C00861 V=800.0 PL=0
MOVL C00862 V=800.0 PL=0
MOVL C00863 V=800.0 PL=0
MOVL C00864 V=800.0 PL=0
MOVL C00865 V=800.0 PL=0
MOVL C00866 V=800.0 PL=0
MOVL C00867 V=800.0 PL=0
MOVL C00868 V=800.0 PL=0
MOVL C00869 V=800.0 PL=0
MOVL C00870 V=800.0 PL=0
MOVL C00871 V=800.0 PL=0
MOVL C00872 V=800.0 PL=0
MOVL C00873 V=800.0 PL=0
MOVL C00874 V=800.0 PL=0
MOVL C00875 V=800.0 PL=0
MOVL C00876 V=800.0 PL=0
MOVL C00877 V=800.0 PL=0
MOVL C00878 V=800.0 PL=0
MOVL C00879 V=800.0 PL=0
MOVL C00880 V=800.0 PL=0
MOVL C00881 V=800.0 PL=0
MOVL C00882 V=800.0 PL=0
MOVL C00883 V=800.0 PL=0
MOVL C00884 V=800.0 PL=0
MOVL C00885 V=800.0 PL=0
MOVL C00886 V=800.0 PL=0
MOVL C00887 V=800.0 PL=0
MOVL C00888 V=800.0 PL=0
MOVL C00889 V=800.0 PL=0
MOVL C00890 V=800.0 PL=0
MOVL C00891 V=800.0 PL=0
MOVL C00892 V=800.0 PL=0
MOVL C00893 V=800.0 PL=0
MOVL C00894 V=800.0 PL=0
MOVL C00895 V=800.0 PL=0
MOVL C00896 V=800.0 PL=0
MOVL C00897 V=800.0 PL=0
MOVL C00898 V=800.0 PL=0
MOVL C00899 V=800.0 PL=0
MOVL C00900 V=800.0 PL=0
MOVL C00901 V=800.0 PL=0
MOVL C00902 V=800.0 PL=0
MOVL C00903 V=800.0 PL=0
MOVL C00904 V=800.0 PL=0
MOVL C00905 V=800.0 PL=0
MOVL C00906 V=800.0 PL=0
MOVL C00907 V=800.0 PL=0
MOVL C00908 V=800.0 PL=0
MOVL C00909 V=800.0 PL=0
MOVL C00910 V=800.0 PL=0
MOVL C00911 V=800.0 PL=0
MOVL C00912 V=800.0 PL=0
MOVL C00913 V=800.0 PL=0
MOVL C00914 V=800.0 PL=0
MOVL C00915 V=800.0 PL=0
MOVL C00916 V=800.0 PL=0
MOVL C00917 V=800.0 PL=0
MOVL C00918 V=800.0 PL=0
MOVL C00919 V=800.0 PL=0
MOVL C00920 V=800.0 PL=0
MOVL C00921 V=800.0 PL=0
MOVL C00922 V=800.0 PL=0
MOVL C00923 V=800.0 PL=0
MOVL C00924 V=800.0 PL=0
MOVL C00925 V=800.0 PL=0
MOVL C00926 V=800.0 PL=0
MOVL C00927 V=800.0 PL=0
MOVL C00928 V=800.0 PL=0
MOVL C00929 V=800.0 PL=0
MOVL C00930 V=800.0 PL=0
MOVL C00931 V=800.0 PL=0
MOVL C00932 V=800.0 PL=0
MOVL C00933 V=800.0 PL=0
MOVL C00934 V=800.0 PL=0
MOVL C00935 V=800.0 PL=0
MOVL C00936 V=800.0 PL=0
MOVL C00937 V=800.0 PL=0
MOVL C00938 V=800.0 PL=0
MOVL C00939 V=800.0 PL=0
MOVL C00940 V=800.0 PL=0
MOVL C00941 V=800.0 PL=0
MOVL C00942 V=800.0 PL=0
MOVL C00943 V=800.0 PL=0
MOVL C00944 V=800.0 PL=0
MOVL C00945 V=800.0 PL=0
MOVL C00946 V=800.0 PL=0
MOVL C00947 V=800.0 PL=0
MOVL C00948 V=800.0 PL=0
MOVL C00949 V=800.0 PL=0
MOVL C00950 V=800.0 PL=0
MOVL C00951 V=800.0 PL=0
MOVL C00952 V=800.0 PL=0
MOVL C00953 V=800.0 PL=0
MOVL C00954 V=800.0 PL=0
MOVL C00955 V=800.0 PL=0
MOVL C00956 V=800.0 PL=0
MOVL C00957 V=800.0 PL=0
MOVL C00958 V=800.0 PL=0
MOVL C00959 V=800.0 PL=0
MOVL C00960 V=800.0 PL=0
MOVL C00961 V=800.0 PL=0
MOVL C00962 V=800.0 PL=0
MOVL C00963 V=800.0 PL=0
MOVL C00964 V=800.0 PL=0
MOVL C00965 V=800.0 PL=0
MOVL C00966 V=800.0 PL=0
MOVL C00967 V=800.0 PL=0
MOVL C00968 V=800.0 PL=0
MOVL C00969 V=800.0 PL=0
MOVL C00970 V=800.0 PL=0
MOVL C00971 V=800.0 PL=0
MOVL C00972 V=800.0 PL=0
MOVL C00973 V=800.0 PL=0
MOVL C00974 V=800.0 PL=0
MOVL C00975 V=800.0 PL=0
MOVL C00976 V=800.0 PL=0
MOVL C00977 V=800.0 PL=0
MOVL C00978 V=800.0 PL=0
MOVL C00979 V=800.0 PL=0
MOVL C00980 V=800.0 PL=0
MOVL C00981 V=800.0 PL=0
MOVL C00982 V=800.0 PL=0
MOVL C00983 V=800.0 PL=0
MOVL C00984 V=800.0 PL=0
MOVL C00985 V=800.0 PL=0
MOVL C00986 V=800.0 PL=0
MOVL C00987 V=800.0 PL=0
MOVL C00988 V=800.0 PL=0
MOVL C00989 V=800.0 PL=0
MOVL C00990 V=800.0 PL=0
MOVL C00991 V=800.0 PL=0
MOVL C00992 V=800.0 PL=0
MOVL C00993 V=800.0 PL=0
MOVL C00994 V=800.0 PL=0
MOVL C00995 V=800.0 PL=0
MOVL C00996 V=800.0 PL=0
MOVL C00997 V=800.0 PL=0
MOVL C00998 V=800.0 PL=0
MOVL C00999 V=800.0 PL=0
MOVL C01000 V=800.0 PL=0
MOVL C01001 V=800.0 PL=0
MOVL C01002 V=800.0 PL=0
MOVL C01003 V=800.0 PL=0
MOVL C01004 V=800.0 PL=0
MOVL C01005 V=800.0 PL=0
MOVL C01006 V=800.0 PL=0
MOVL C01007 V=800.0 PL=0
MOVL C01008 V=800.0 PL=0
MOVL C01009 V=800.0 PL=0
MOVL C01010 V=800.0 PL=0
MOVL C01011 V=800.0 PL=0
MOVL C01012 V=800.0 PL=0
MOVL C01013 V=800.0 PL=0
MOVL C01014 V=800.0 PL=0
MOVL C01015 V=800.0 PL=0
MOVL C01016 V=800.0 PL=0
MOVL C01017 V=800.0 PL=0
MOVL C01018 V=800.0 PL=0
MOVL C01019 V=800.0 PL=0
MOVL C01020 V=800.0 PL=0
MOVL C01021 V=800.0 PL=0
MOVL C01022 V=800.0 PL=0
MOVL C01023 V=800.0 PL=0
MOVL C01024 V=800.0 PL=0
MOVL C01025 V=800.0 PL=0
MOVL C01026 V=800.0 PL=0
MOVL C01027 V=800.0 PL=0
MOVL C01028 V=800.0 PL=0
MOVL C01029 V=800.0 PL=0
MOVL C01030 V=800.0 PL=0
MOVL C01031 V=800.0 PL=0
MOVL C01032 V=800.0 PL=0
MOVL C01033 V=800.0 PL=0
MOVL C01034 V=800.0 PL=0
MOVL C01035 V=800.0 PL=0
MOVL C01036 V=800.0 PL=0
MOVL C01037 V=800.0 PL=0
MOVL C01038 V=800.0 PL=0
MOVL C01039 V=800.0 PL=0
MOVL C01040 V=800.0 PL=0
MOVL C01041 V=800.0 PL=0
MOVL C01042 V=800.0 PL=0
MOVL C01043 V=800.0 PL=0
MOVL C01044 V=800.0 PL=0
MOVL C01045 V=800.0 PL=0
MOVL C01046 V=800.0 PL=0
MOVL C01047 V=800.0 PL=0
MOVL C01048 V=800.0 PL=0
MOVL C01049 V=800.0 PL=0
MOVL C01050 V=800.0 PL=0
MOVL C01051 V=800.0 PL=0
MOVL C01052 V=800.0 PL=0
MOVL C01053 V=800.0 PL=0
MOVL C01054 V=800.0 PL=0
MOVL C01055 V=800.0 PL=0
MOVL C01056 V=800.0 PL=0
MOVL C01057 V=800.0 PL=0
MOVL C01058 V=800.0 PL=0
MOVL C01059 V=800.0 PL=0
MOVL C01060 V=800.0 PL=0
MOVL C01061 V=800.0 PL=0
MOVL C01062 V=800.0 PL=0
MOVL C01063 V=800.0 PL=0
MOVL C01064 V=800.0 PL=0
MOVL C01065 V=800.0 PL=0
MOVL C01066 V=800.0 PL=0
MOVL C01067 V=800.0 PL=0
MOVL C01068 V=800.0 PL=0
MOVL C01069 V=800.0 PL=0
MOVL C01070 V=800.0 PL=0
MOVL C01071 V=800.0 PL=0
MOVL C01072 V=800.0 PL=0
MOVL C01073 V=800.0 PL=0
MOVL C01074 V=800.0 PL=0
MOVL C01075 V=800.0 PL=0
MOVL C01076 V=800.0 PL=0
MOVL C01077 V=800.0 PL=0
MOVL C01078 V=800.0 PL=0
MOVL C01079 V=800.0 PL=0
MOVL C01080 V=800.0 PL=0
MOVL C01081 V=800.0 PL=0
MOVL C01082 V=800.0 PL=0
MOVL C01083 V=800.0 PL=0
MOVL C01084 V=800.0 PL=0
MOVL C01085 V=800.0 PL=0
MOVL C01086 V=800.0 PL=0
MOVL C01087 V=800.0 PL=0
MOVL C01088 V=800.0 PL=0
MOVL C01089 V=800.0 PL=0
MOVL C01090 V=800.0 PL=0
MOVL C01091 V=800.0 PL=0
MOVL C01092 V=800.0 PL=0
MOVL C01093 V=800.0 PL=0
MOVL C01094 V=800.0 PL=0
MOVL C01095 V=800.0 PL=0
MOVL C01096 V=800.0 PL=0
MOVL C01097 V=800.0 PL=0
MOVL C01098 V=800.0 PL=0
MOVL C01099 V=800.0 PL=0
MOVL C01100 V=800.0 PL=0
MOVL C01101 V=800.0 PL=0
MOVL C01102 V=800.0 PL=0
MOVL C01103 V=800.0 PL=0
MOVL C01104 V=800.0 PL=0
MOVL C01105 V=800.0 PL=0
MOVL C01106 V=800.0 PL=0
MOVL C01107 V=800.0 PL=0
MOVL C01108 V=800.0 PL=0
MOVL C01109 V=800.0 PL=0
MOVL C01110 V=800.0 PL=0
MOVL C01111 V=800.0 PL=0
MOVL C01112 V=800.0 PL=0
MOVL C01113 V=800.0 PL=0
MOVL C01114 V=800.0 PL=0
MOVL C01115 V=800.0 PL=0
MOVL C01116 V=800.0 PL=0
MOVL C01117 V=800.0 PL=0
MOVL C01118 V=800.0 PL=0
MOVL C01119 V=800.0 PL=0
MOVL C01120 V=800.0 PL=0
MOVL C01121 V=800.0 PL=0
MOVL C01122 V=800.0 PL=0
MOVL C01123 V=800.0 PL=0
MOVL C01124 V=800.0 PL=0
MOVL C01125 V=800.0 PL=0
MOVL C01126 V=800.0 PL=0
MOVL C01127 V=800.0 PL=0
MOVL C01128 V=800.0 PL=0
MOVL C01129 V=800.0 PL=0
MOVL C01130 V=800.0 PL=0
MOVL C01131 V=800.0 PL=0
MOVL C01132 V=800.0 PL=0
MOVL C01133 V=800.0 PL=0
MOVL C01134 V=800.0 PL=0
MOVL C01135 V=800.0 PL=0
MOVL C01136 V=800.0 PL=0
MOVL C01137 V=800.0 PL=0
MOVL C01138 V=800.0 PL=0
MOVL C01139 V=800.0 PL=0
MOVL C01140 V=800.0 PL=0
MOVL C01141 V=800.0 PL=0
MOVL C01142 V=800.0 PL=0
MOVL C01143 V=800.0 PL=0
MOVL C01144 V=800.0 PL=0
MOVL C01145 V=800.0 PL=0
MOVL C01146 V=800.0 PL=0
MOVL C01147 V=800.0 PL=0
MOVL C01148 V=800.0 PL=0
MOVL C01149 V=800.0 PL=0
MOVL C01150 V=800.0 PL=0
MOVL C01151 V=800.0 PL=0
MOVL C01152 V=800.0 PL=0
MOVL C01153 V=800.0 PL=0
MOVL C01154 V=800.0 PL=0
MOVL C01155 V=800.0 PL=0
MOVL C01156 V=800.0 PL=0
MOVL C01157 V=800.0 PL=0
MOVL C01158 V=800.0 PL=0
MOVL C01159 V=800.0 PL=0
MOVL C01160 V=800.0 PL=0
MOVL C01161 V=800.0 PL=0
MOVL C01162 V=800.0 PL=0
MOVL C01163 V=800.0 PL=0
MOVL C01164 V=800.0 PL=0
MOVL C01165 V=800.0 PL=0
MOVL C01166 V=800.0 PL=0
MOVL C01167 V=800.0 PL=0
MOVL C01168 V=800.0 PL=0
MOVL C01169 V=800.0 PL=0
MOVL C01170 V=800.0 PL=0
MOVL C01171 V=800.0 PL=0
MOVL C01172 V=800.0 PL=0
MOVL C01173 V=800.0 PL=0
MOVL C01174 V=800.0 PL=0
MOVL C01175 V=800.0 PL=0
MOVL C01176 V=800.0 PL=0
MOVL C01177 V=800.0 PL=0
MOVL C01178 V=800.0 PL=0
MOVL C01179 V=800.0 PL=0
MOVL C01180 V=800.0 PL=0
MOVL C01181 V=800.0 PL=0
MOVL C01182 V=800.0 PL=0
MOVL C01183 V=800.0 PL=0
MOVL C01184 V=800.0 PL=0
MOVL C01185 V=800.0 PL=0
MOVL C01186 V=800.0 PL=0
MOVL C01187 V=800.0 PL=0
MOVL C01188 V=800.0 PL=0
MOVL C01189 V=800.0 PL=0
MOVL C01190 V=800.0 PL=0
MOVL C01191 V=800.0 PL=0
MOVL C01192 V=800.0 PL=0
MOVL C01193 V=800.0 PL=0
MOVL C01194 V=800.0 PL=0
MOVL C01195 V=800.0 PL=0
MOVL C01196 V=800.0 PL=0
MOVL C01197 V=800.0 PL=0
MOVL C01198 V=800.0 PL=0
MOVL C01199 V=800.0 PL=0
MOVL C01200 V=800.0 PL=0
MOVL C01201 V=800.0 PL=0
MOVL C01202 V=800.0 PL=0
MOVL C01203 V=800.0 PL=0
MOVL C01204 V=800.0 PL=0
MOVL C01205 V=800.0 PL=0
MOVL C01206 V=800.0 PL=0
MOVL C01207 V=800.0 PL=0
MOVL C01208 V=800.0 PL=0
MOVL C01209 V=800.0 PL=0
MOVL C01210 V=800.0 PL=0
MOVL C01211 V=800.0 PL=0
MOVL C01212 V=800.0 PL=0
MOVL C01213 V=800.0 PL=0
MOVL C01214 V=800.0 PL=0
MOVL C01215 V=800.0 PL=0
MOVL C01216 V=800.0 PL=0
MOVL C01217 V=800.0 PL=0
MOVL C01218 V=800.0 PL=0
MOVL C01219 V=800.0 PL=0
MOVL C01220 V=800.0 PL=0
MOVL C01221 V=800.0 PL=0
MOVL C01222 V=800.0 PL=0
MOVL C01223 V=800.0 PL=0
MOVL C01224 V=800.0 PL=0
MOVL C01225 V=800.0 PL=0
MOVL C01226 V=800.0 PL=0
MOVL C01227 V=800.0 PL=0
MOVL C01228 V=800.0 PL=0
MOVL C01229 V=800.0 PL=0
MOVL C01230 V=800.0 PL=0
MOVL C01231 V=800.0 PL=0
MOVL C01232 V=800.0 PL=0
MOVL C01233 V=800.0 PL=0
MOVL C01234 V=800.0 PL=0
MOVL C01235 V=800.0 PL=0
MOVL C01236 V=800.0 PL=0
MOVL C01237 V=800.0 PL=0
MOVL C01238 V=800.0 PL=0
MOVL C01239 V=800.0 PL=0
MOVL C01240 V=800.0 PL=0
MOVL C01241 V=800.0 PL=0
MOVL C01242 V=800.0 PL=0
MOVL C01243 V=800.0 PL=0
MOVL C01244 V=800.0 PL=0
MOVL C01245 V=800.0 PL=0
MOVL C01246 V=800.0 PL=0
MOVL C01247 V=800.0 PL=0
MOVL C01248 V=800.0 PL=0
MOVL C01249 V=800.0 PL=0
MOVL C01250 V=800.0 PL=0
MOVL C01251 V=800.0 PL=0
MOVL C01252 V=800.0 PL=0
MOVL C01253 V=800.0 PL=0
MOVL C01254 V=800.0 PL=0
MOVL C01255 V=800.0 PL=0
MOVL C01256 V=800.0 PL=0
MOVL C01257 V=800.0 PL=0
MOVL C01258 V=800.0 PL=0
MOVL C01259 V=800.0 PL=0
MOVL C01260 V=800.0 PL=0
MOVL C01261 V=800.0 PL=0
MOVL C01262 V=800.0 PL=0
MOVL C01263 V=800.0 PL=0
MOVL C01264 V=800.0 PL=0
MOVL C01265 V=800.0 PL=0
MOVL C01266 V=800.0 PL=0
MOVL C01267 V=800.0 PL=0
MOVL C01268 V=800.0 PL=0
MOVL C01269 V=800.0 PL=0
MOVL C01270 V=800.0 PL=0
MOVL C01271 V=800.0 PL=0
MOVL C01272 V=800.0 PL=0
MOVL C01273 V=800.0 PL=0
MOVL C01274 V=800.0 PL=0
MOVL C01275 V=800.0 PL=0
MOVL C01276 V=800.0 PL=0
MOVL C01277 V=800.0 PL=0
MOVL C01278 V=800.0 PL=0
MOVL C01279 V=800.0 PL=0
MOVL C01280 V=800.0 PL=0
MOVL C01281 V=800.0 PL=0
MOVL C01282 V=800.0 PL=0
MOVL C01283 V=800.0 PL=0
MOVL C01284 V=800.0 PL=0
MOVL C01285 V=800.0 PL=0
MOVL C01286 V=800.0 PL=0
MOVL C01287 V=800.0 PL=0
MOVL C01288 V=800.0 PL=0
MOVL C01289 V=800.0 PL=0
MOVL C01290 V=800.0 PL=0
MOVL C01291 V=800.0 PL=0
MOVL C01292 V=800.0 PL=0
MOVL C01293 V=800.0 PL=0
MOVL C01294 V=800.0 PL=0
MOVL C01295 V=800.0 PL=0
MOVL C01296 V=800.0 PL=0
MOVL C01297 V=800.0 PL=0
MOVL C01298 V=800.0 PL=0
MOVL C01299 V=800.0 PL=0
MOVL C01300 V=800.0 PL=0
MOVL C01301 V=800.0 PL=0
MOVL C01302 V=800.0 PL=0
MOVL C01303 V=800.0 PL=0
MOVL C01304 V=800.0 PL=0
MOVL C01305 V=800.0 PL=0
MOVL C01306 V=800.0 PL=0
MOVL C01307 V=800.0 PL=0
MOVL C01308 V=800.0 PL=0
MOVL C01309 V=800.0 PL=0
MOVL C01310 V=800.0 PL=0
MOVL C01311 V=800.0 PL=0
MOVL C01312 V=800.0 PL=0
MOVL C01313 V=800.0 PL=0
MOVL C01314 V=800.0 PL=0
MOVL C01315 V=800.0 PL=0
MOVL C01316 V=800.0 PL=0
MOVL C01317 V=800.0 PL=0
MOVL C01318 V=800.0 PL=0
MOVL C01319 V=800.0 PL=0
MOVL C01320 V=800.0 PL=0
MOVL C01321 V=800.0 PL=0
MOVL C01322 V=800.0 PL=0
MOVL C01323 V=800.0 PL=0
MOVL C01324 V=800.0 PL=0
MOVL C01325 V=800.0 PL=0
MOVL C01326 V=800.0 PL=0
MOVL C01327 V=800.0 PL=0
MOVL C01328 V=800.0 PL=0
MOVL C01329 V=800.0 PL=0
MOVL C01330 V=800.0 PL=0
MOVL C01331 V=800.0 PL=0
MOVL C01332 V=800.0 PL=0
MOVL C01333 V=800.0 PL=0
MOVL C01334 V=800.0 PL=0
MOVL C01335 V=800.0 PL=0
MOVL C01336 V=800.0 PL=0
MOVL C01337 V=800.0 PL=0
MOVL C01338 V=800.0 PL=0
MOVL C01339 V=800.0 PL=0
MOVL C01340 V=800.0 PL=0
MOVL C01341 V=800.0 PL=0
MOVL C01342 V=800.0 PL=0
MOVL C01343 V=800.0 PL=0
MOVL C01344 V=800.0 PL=0
MOVL C01345 V=800.0 PL=0
MOVL C01346 V=800.0 PL=0
MOVL C01347 V=800.0 PL=0
MOVL C01348 V=800.0 PL=0
MOVL C01349 V=800.0 PL=0
MOVL C01350 V=800.0 PL=0
MOVL C01351 V=800.0 PL=0
MOVL C01352 V=800.0 PL=0
MOVL C01353 V=800.0 PL=0
MOVL C01354 V=800.0 PL=0
MOVL C01355 V=800.0 PL=0
MOVL C01356 V=800.0 PL=0
MOVL C01357 V=800.0 PL=0
MOVL C01358 V=800.0 PL=0
MOVL C01359 V=800.0 PL=0
MOVL C01360 V=800.0 PL=0
MOVL C01361 V=800.0 PL=0
MOVL C01362 V=800.0 PL=0
MOVL C01363 V=800.0 PL=0
MOVL C01364 V=800.0 PL=0
MOVL C01365 V=800.0 PL=0
MOVL C01366 V=800.0 PL=0
MOVL C01367 V=800.0 PL=0
MOVL C01368 V=800.0 PL=0
MOVL C01369 V=800.0 PL=0
MOVL C01370 V=800.0 PL=0
MOVL C01371 V=800.0 PL=0
MOVL C01372 V=800.0 PL=0
MOVL C01373 V=800.0 PL=0
MOVL C01374 V=800.0 PL=0
MOVL C01375 V=800.0 PL=0
MOVL C01376 V=800.0 PL=0
MOVL C01377 V=800.0 PL=0
MOVL C01378 V=800.0 PL=0
MOVL C01379 V=800.0 PL=0
MOVL C01380 V=800.0 PL=0
MOVL C01381 V=800.0 PL=0
MOVL C01382 V=800.0 PL=0
MOVL C01383 V=800.0 PL=0
MOVL C01384 V=800.0 PL=0
MOVL C01385 V=800.0 PL=0
MOVL C01386 V=800.0 PL=0
MOVL C01387 V=800.0 PL=0
MOVL C01388 V=800.0 PL=0
MOVL C01389 V=800.0 PL=0
MOVL C01390 V=800.0 PL=0
MOVL C01391 V=800.0 PL=0
MOVL C01392 V=800.0 PL=0
MOVL C01393 V=800.0 PL=0
MOVL C01394 V=800.0 PL=0
MOVL C01395 V=800.0 PL=0
MOVL C01396 V=800.0 PL=0
MOVL C01397 V=800.0 PL=0
MOVL C01398 V=800.0 PL=0
MOVL C01399 V=800.0 PL=0
MOVL C01400 V=800.0 PL=0
MOVL C01401 V=800.0 PL=0
MOVL C01402 V=800.0 PL=0
MOVL C01403 V=800.0 PL=0
MOVL C01404 V=800.0 PL=0
MOVL C01405 V=800.0 PL=0
MOVL C01406 V=800.0 PL=0
MOVL C01407 V=800.0 PL=0
MOVL C01408 V=800.0 PL=0
MOVL C01409 V=800.0 PL=0
MOVL C01410 V=800.0 PL=0
MOVL C01411 V=800.0 PL=0
MOVL C01412 V=800.0 PL=0
MOVL C01413 V=800.0 PL=0
MOVL C01414 V=800.0 PL=0
MOVL C01415 V=800.0 PL=0
MOVL C01416 V=800.0 PL=0
MOVL C01417 V=800.0 PL=0
MOVL C01418 V=800.0 PL=0
MOVL C01419 V=800.0 PL=0
MOVL C01420 V=800.0 PL=0
MOVL C01421 V=800.0 PL=0
MOVL C01422 V=800.0 PL=0
MOVL C01423 V=800.0 PL=0
MOVL C01424 V=800.0 PL=0
MOVL C01425 V=800.0 PL=0
MOVL C01426 V=800.0 PL=0
MOVL C01427 V=800.0 PL=0
MOVL C01428 V=800.0 PL=0
MOVL C01429 V=800.0 PL=0
MOVL C01430 V=800.0 PL=0
MOVL C01431 V=800.0 PL=0
MOVL C01432 V=800.0 PL=0
MOVL C01433 V=800.0 PL=0
MOVL C01434 V=800.0 PL=0
MOVL C01435 V=800.0 PL=0
MOVL C01436 V=800.0 PL=0
MOVL C01437 V=800.0 PL=0
MOVL C01438 V=800.0 PL=0
MOVL C01439 V=800.0 PL=0
MOVL C01440 V=800.0 PL=0
MOVL C01441 V=800.0 PL=0
MOVL C01442 V=800.0 PL=0
MOVL C01443 V=800.0 PL=0
MOVL C01444 V=800.0 PL=0
MOVL C01445 V=800.0 PL=0
MOVL C01446 V=800.0 PL=0
MOVL C01447 V=800.0 PL=0
MOVL C01448 V=800.0 PL=0
MOVL C01449 V=800.0 PL=0
MOVL C01450 V=800.0 PL=0
MOVL C01451 V=800.0 PL=0
MOVL C01452 V=800.0 PL=0
MOVL C01453 V=800.0 PL=0
MOVL C01454 V=800.0 PL=0
MOVL C01455 V=800.0 PL=0
MOVL C01456 V=800.0 PL=0
MOVL C01457 V=800.0 PL=0
MOVL C01458 V=800.0 PL=0
MOVL C01459 V=800.0 PL=0
MOVL C01460 V=800.0 PL=0
MOVL C01461 V=800.0 PL=0
MOVL C01462 V=800.0 PL=0
MOVL C01463 V=800.0 PL=0
MOVL C01464 V=800.0 PL=0
MOVL C01465 V=800.0 PL=0
MOVL C01466 V=800.0 PL=0
MOVL C01467 V=800.0 PL=0
MOVL C01468 V=800.0 PL=0
MOVL C01469 V=800.0 PL=0
MOVL C01470 V=800.0 PL=0
MOVL C01471 V=800.0 PL=0
MOVL C01472 V=800.0 PL=0
MOVL C01473 V=800.0 PL=0
MOVL C01474 V=800.0 PL=0
MOVL C01475 V=800.0 PL=0
MOVL C01476 V=800.0 PL=0
MOVL C01477 V=800.0 PL=0
MOVL C01478 V=800.0 PL=0
MOVL C01479 V=800.0 PL=0
MOVL C01480 V=800.0 PL=0
MOVL C01481 V=800.0 PL=0
MOVL C01482 V=800.0 PL=0
MOVL C01483 V=800.0 PL=0
MOVL C01484 V=800.0 PL=0
MOVL C01485 V=800.0 PL=0
MOVL C01486 V=800.0 PL=0
MOVL C01487 V=800.0 PL=0
MOVL C01488 V=800.0 PL=0
MOVL C01489 V=800.0 PL=0
MOVL C01490 V=800.0 PL=0
MOVL C01491 V=800.0 PL=0
MOVL C01492 V=800.0 PL=0
MOVL C01493 V=800.0 PL=0
MOVL C01494 V=800.0 PL=0
MOVL C01495 V=800.0 PL=0
MOVL C01496 V=800.0 PL=0
MOVL C01497 V=800.0 PL=0
MOVL C01498 V=800.0 PL=0
MOVL C01499 V=800.0 PL=0
MOVL C01500 V=800.0 PL=0
MOVL C01501 V=800.0 PL=0
MOVL C01502 V=800.0 PL=0
MOVL C01503 V=800.0 PL=0
MOVL C01504 V=800.0 PL=0
MOVL C01505 V=800.0 PL=0
MOVL C01506 V=800.0 PL=0
MOVL C01507 V=800.0 PL=0
MOVL C01508 V=800.0 PL=0
MOVL C01509 V=800.0 PL=0
MOVL C01510 V=800.0 PL=0
MOVL C01511 V=800.0 PL=0
MOVL C01512 V=800.0 PL=0
MOVL C01513 V=800.0 PL=0
MOVL C01514 V=800.0 PL=0
MOVL C01515 V=800.0 PL=0
MOVL C01516 V=800.0 PL=0
MOVL C01517 V=800.0 PL=0
MOVL C01518 V=800.0 PL=0
MOVL C01519 V=800.0 PL=0
MOVL C01520 V=800.0 PL=0
MOVL C01521 V=800.0 PL=0
MOVL C01522 V=800.0 PL=0
MOVL C01523 V=800.0 PL=0
MOVL C01524 V=800.0 PL=0
MOVL C01525 V=800.0 PL=0
MOVL C01526 V=800.0 PL=0
MOVL C01527 V=800.0 PL=0
MOVL C01528 V=800.0 PL=0
MOVL C01529 V=800.0 PL=0
MOVL C01530 V=800.0 PL=0
MOVL C01531 V=800.0 PL=0
MOVL C01532 V=800.0 PL=0
MOVL C01533 V=800.0 PL=0
MOVL C01534 V=800.0 PL=0
MOVL C01535 V=800.0 PL=0
MOVL C01536 V=800.0 PL=0
MOVL C01537 V=800.0 PL=0
MOVL C01538 V=800.0 PL=0
MOVL C01539 V=800.0 PL=0
MOVL C01540 V=800.0 PL=0
MOVL C01541 V=800.0 PL=0
MOVL C01542 V=800.0 PL=0
MOVL C01543 V=800.0 PL=0
MOVL C01544 V=800.0 PL=0
MOVL C01545 V=800.0 PL=0
MOVL C01546 V=800.0 PL=0
MOVL C01547 V=800.0 PL=0
MOVL C01548 V=800.0 PL=0
MOVL C01549 V=800.0 PL=0
MOVL C01550 V=800.0 PL=0
MOVL C01551 V=800.0 PL=0
MOVL C01552 V=800.0 PL=0
MOVL C01553 V=800.0 PL=0
MOVL C01554 V=800.0 PL=0
MOVL C01555 V=800.0 PL=0
MOVL C01556 V=800.0 PL=0
MOVL C01557 V=800.0 PL=0
MOVL C01558 V=800.0 PL=0
MOVL C01559 V=800.0 PL=0
MOVL C01560 V=800.0 PL=0
MOVL C01561 V=800.0 PL=0
MOVL C01562 V=800.0 PL=0
MOVL C01563 V=800.0 PL=0
MOVL C01564 V=800.0 PL=0
MOVL C01565 V=800.0 PL=0
MOVL C01566 V=800.0 PL=0
MOVL C01567 V=800.0 PL=0
MOVL C01568 V=800.0 PL=0
MOVL C01569 V=800.0 PL=0
MOVL C01570 V=800.0 PL=0
MOVL C01571 V=800.0 PL=0
MOVL C01572 V=800.0 PL=0
MOVL C01573 V=800.0 PL=0
MOVL C01574 V=800.0 PL=0
MOVL C01575 V=800.0 PL=0
MOVL C01576 V=800.0 PL=0
MOVL C01577 V=800.0 PL=0
MOVL C01578 V=800.0 PL=0
MOVL C01579 V=800.0 PL=0
MOVL C01580 V=800.0 PL=0
MOVL C01581 V=800.0 PL=0
MOVL C01582 V=800.0 PL=0
MOVL C01583 V=800.0 PL=0
MOVL C01584 V=800.0 PL=0
MOVL C01585 V=800.0 PL=0
MOVL C01586 V=800.0 PL=0
MOVL C01587 V=800.0 PL=0
MOVL C01588 V=800.0 PL=0
MOVL C01589 V=800.0 PL=0
MOVL C01590 V=800.0 PL=0
MOVL C01591 V=800.0 PL=0
MOVL C01592 V=800.0 PL=0
MOVL C01593 V=800.0 PL=0
MOVL C01594 V=800.0 PL=0
MOVL C01595 V=800.0 PL=0
MOVL C01596 V=800.0 PL=0
MOVL C01597 V=800.0 PL=0
MOVL C01598 V=800.0 PL=0
MOVL C01599 V=800.0 PL=0
MOVL C01600 V=800.0 PL=0
MOVL C01601 V=800.0 PL=0
MOVL C01602 V=800.0 PL=0
MOVL C01603 V=800.0 PL=0
MOVL C01604 V=800.0 PL=0
MOVL C01605 V=800.0 PL=0
MOVL C01606 V=800.0 PL=0
MOVL C01607 V=800.0 PL=0
MOVL C01608 V=800.0 PL=0
MOVL C01609 V=800.0 PL=0
MOVL C01610 V=800.0 PL=0
MOVL C01611 V=800.0 PL=0
MOVL C01612 V=800.0 PL=0
MOVL C01613 V=800.0 PL=0
MOVL C01614 V=800.0 PL=0
MOVL C01615 V=800.0 PL=0
MOVL C01616 V=800.0 PL=0
MOVL C01617 V=800.0 PL=0
MOVL C01618 V=800.0 PL=0
MOVL C01619 V=800.0 PL=0
MOVL C01620 V=800.0 PL=0
MOVL C01621 V=800.0 PL=0
MOVL C01622 V=800.0 PL=0
MOVL C01623 V=800.0 PL=0
MOVL C01624 V=800.0 PL=0
MOVL C01625 V=800.0 PL=0
MOVL C01626 V=800.0 PL=0
MOVL C01627 V=800.0 PL=0
MOVL C01628 V=800.0 PL=0
MOVL C01629 V=800.0 PL=0
MOVL C01630 V=800.0 PL=0
MOVL C01631 V=800.0 PL=0
MOVL C01632 V=800.0 PL=0
MOVL C01633 V=800.0 PL=0
MOVL C01634 V=800.0 PL=0
MOVL C01635 V=800.0 PL=0
MOVL C01636 V=800.0 PL=0
MOVL C01637 V=800.0 PL=0
MOVL C01638 V=800.0 PL=0
MOVL C01639 V=800.0 PL=0
MOVL C01640 V=800.0 PL=0
MOVL C01641 V=800.0 PL=0
MOVL C01642 V=800.0 PL=0
MOVL C01643 V=800.0 PL=0
MOVL C01644 V=800.0 PL=0
MOVL C01645 V=800.0 PL=0
MOVL C01646 V=800.0 PL=0
MOVL C01647 V=800.0 PL=0
MOVL C01648 V=800.0 PL=0
MOVL C01649 V=800.0 PL=0
MOVL C01650 V=800.0 PL=0
MOVL C01651 V=800.0 PL=0
MOVL C01652 V=800.0 PL=0
MOVL C01653 V=800.0 PL=0
MOVL C01654 V=800.0 PL=0
MOVL C01655 V=800.0 PL=0
MOVL C01656 V=800.0 PL=0
MOVL C01657 V=800.0 PL=0
MOVL C01658 V=800.0 PL=0
MOVL C01659 V=800.0 PL=0
MOVL C01660 V=800.0 PL=0
MOVL C01661 V=800.0 PL=0
MOVL C01662 V=800.0 PL=0
MOVL C01663 V=800.0 PL=0
MOVL C01664 V=800.0 PL=0
MOVL C01665 V=800.0 PL=0
MOVL C01666 V=800.0 PL=0
MOVL C01667 V=800.0 PL=0
MOVL C01668 V=800.0 PL=0
MOVL C01669 V=800.0 PL=0
MOVL C01670 V=800.0 PL=0
MOVL C01671 V=800.0 PL=0
MOVL C01672 V=800.0 PL=0
MOVL C01673 V=800.0 PL=0
MOVL C01674 V=800.0 PL=0
MOVL C01675 V=800.0 PL=0
MOVL C01676 V=800.0 PL=0
MOVL C01677 V=800.0 PL=0
MOVL C01678 V=800.0 PL=0
MOVL C01679 V=800.0 PL=0
MOVL C01680 V=800.0 PL=0
MOVL C01681 V=800.0 PL=0
MOVL C01682 V=800.0 PL=0
MOVL C01683 V=800.0 PL=0
MOVL C01684 V=800.0 PL=0
MOVL C01685 V=800.0 PL=0
MOVL C01686 V=800.0 PL=0
MOVL C01687 V=800.0 PL=0
MOVL C01688 V=800.0 PL=0
MOVL C01689 V=800.0 PL=0
MOVL C01690 V=800.0 PL=0
MOVL C01691 V=800.0 PL=0
MOVL C01692 V=800.0 PL=0
MOVL C01693 V=800.0 PL=0
MOVL C01694 V=800.0 PL=0
MOVL C01695 V=800.0 PL=0
MOVL C01696 V=800.0 PL=0
MOVL C01697 V=800.0 PL=0
MOVL C01698 V=800.0 PL=0
MOVL C01699 V=800.0 PL=0
MOVL C01700 V=800.0 PL=0
MOVL C01701 V=800.0 PL=0
MOVL C01702 V=800.0 PL=0
MOVL C01703 V=800.0 PL=0
MOVL C01704 V=800.0 PL=0
MOVL C01705 V=800.0 PL=0
MOVL C01706 V=800.0 PL=0
MOVL C01707 V=800.0 PL=0
MOVL C01708 V=800.0 PL=0
MOVL C01709 V=800.0 PL=0
MOVL C01710 V=800.0 PL=0
MOVL C01711 V=800.0 PL=0
MOVL C01712 V=800.0 PL=0
MOVL C01713 V=800.0 PL=0
MOVL C01714 V=800.0 PL=0
MOVL C01715 V=800.0 PL=0
MOVL C01716 V=800.0 PL=0
MOVL C01717 V=800.0 PL=0
MOVL C01718 V=800.0 PL=0
MOVL C01719 V=800.0 PL=0
MOVL C01720 V=800.0 PL=0
MOVL C01721 V=800.0 PL=0
MOVL C01722 V=800.0 PL=0
MOVL C01723 V=800.0 PL=0
MOVL C01724 V=800.0 PL=0
MOVL C01725 V=800.0 PL=0
MOVL C01726 V=800.0 PL=0
MOVL C01727 V=800.0 PL=0
MOVL C01728 V=800.0 PL=0
MOVL C01729 V=800.0 PL=0
MOVL C01730 V=800.0 PL=0
MOVL C01731 V=800.0 PL=0
MOVL C01732 V=800.0 PL=0
MOVL C01733 V=800.0 PL=0
MOVL C01734 V=800.0 PL=0
MOVL C01735 V=800.0 PL=0
MOVL C01736 V=800.0 PL=0
MOVL C01737 V=800.0 PL=0
MOVL C01738 V=800.0 PL=0
MOVL C01739 V=800.0 PL=0
MOVL C01740 V=800.0 PL=0
MOVL C01741 V=800.0 PL=0
MOVL C01742 V=800.0 PL=0
MOVL C01743 V=800.0 PL=0
MOVL C01744 V=800.0 PL=0
MOVL C01745 V=800.0 PL=0
MOVL C01746 V=800.0 PL=0
MOVL C01747 V=800.0 PL=0
MOVL C01748 V=800.0 PL=0
MOVL C01749 V=800.0 PL=0
MOVL C01750 V=800.0 PL=0
MOVL C01751 V=800.0 PL=0
MOVL C01752 V=800.0 PL=0
MOVL C01753 V=800.0 PL=0
MOVL C01754 V=800.0 PL=0
MOVL C01755 V=800.0 PL=0
MOVL C01756 V=800.0 PL=0
MOVL C01757 V=800.0 PL=0
MOVL C01758 V=800.0 PL=0
MOVL C01759 V=800.0 PL=0
MOVL C01760 V=800.0 PL=0
MOVL C01761 V=800.0 PL=0
MOVL C01762 V=800.0 PL=0
MOVL C01763 V=800.0 PL=0
MOVL C01764 V=800.0 PL=0
MOVL C01765 V=800.0 PL=0
MOVL C01766 V=800.0 PL=0
MOVL C01767 V=800.0 PL=0
MOVL C01768 V=800.0 PL=0
MOVL C01769 V=800.0 PL=0
MOVL C01770 V=800.0 PL=0
MOVL C01771 V=800.0 PL=0
MOVL C01772 V=800.0 PL=0
MOVL C01773 V=800.0 PL=0
MOVL C01774 V=800.0 PL=0
MOVL C01775 V=800.0 PL=0
MOVL C01776 V=800.0 PL=0
MOVL C01777 V=800.0 PL=0
MOVL C01778 V=800.0 PL=0
MOVL C01779 V=800.0 PL=0
MOVL C01780 V=800.0 PL=0
MOVL C01781 V=800.0 PL=0
MOVL C01782 V=800.0 PL=0
MOVL C01783 V=800.0 PL=0
MOVL C01784 V=800.0 PL=0
MOVL C01785 V=800.0 PL=0
MOVL C01786 V=800.0 PL=0
MOVL C01787 V=800.0 PL=0
MOVL C01788 V=800.0 PL=0
MOVL C01789 V=800.0 PL=0
MOVL C01790 V=800.0 PL=0
MOVL C01791 V=800.0 PL=0
MOVL C01792 V=800.0 PL=0
MOVL C01793 V=800.0 PL=0
MOVL C01794 V=800.0 PL=0
MOVL C01795 V=800.0 PL=0
MOVL C01796 V=800.0 PL=0
MOVL C01797 V=800.0 PL=0
MOVL C01798 V=800.0 PL=0
MOVL C01799 V=800.0 PL=0
MOVL C01800 V=800.0 PL=0
MOVL C01801 V=800.0 PL=0
MOVL C01802 V=800.0 PL=0
MOVL C01803 V=800.0 PL=0
MOVL C01804 V=800.0 PL=0
MOVL C01805 V=800.0 PL=0
MOVL C01806 V=800.0 PL=0
MOVL C01807 V=800.0 PL=0
MOVL C01808 V=800.0 PL=0
MOVL C01809 V=800.0 PL=0
MOVL C01810 V=800.0 PL=0
MOVL C01811 V=800.0 PL=0
MOVL C01812 V=800.0 PL=0
MOVL C01813 V=800.0 PL=0
MOVL C01814 V=800.0 PL=0
MOVL C01815 V=800.0 PL=0
MOVL C01816 V=800.0 PL=0
MOVL C01817 V=800.0 PL=0
MOVL C01818 V=800.0 PL=0
MOVL C01819 V=800.0 PL=0
MOVL C01820 V=800.0 PL=0
MOVL C01821 V=800.0 PL=0
MOVL C01822 V=800.0 PL=0
MOVL C01823 V=800.0 PL=0
MOVL C01824 V=800.0 PL=0
MOVL C01825 V=800.0 PL=0
MOVL C01826 V=800.0 PL=0
MOVL C01827 V=800.0 PL=0
MOVL C01828 V=800.0 PL=0
MOVL C01829 V=800.0 PL=0
MOVL C01830 V=800.0 PL=0
MOVL C01831 V=800.0 PL=0
MOVL C01832 V=800.0 PL=0
MOVL C01833 V=800.0 PL=0
MOVL C01834 V=800.0 PL=0
MOVL C01835 V=800.0 PL=0
MOVL C01836 V=800.0 PL=0
MOVL C01837 V=800.0 PL=0
MOVL C01838 V=800.0 PL=0
MOVL C01839 V=800.0 PL=0
MOVL C01840 V=800.0 PL=0
MOVL C01841 V=800.0 PL=0
MOVL C01842 V=800.0 PL=0
MOVL C01843 V=800.0 PL=0
MOVL C01844 V=800.0 PL=0
MOVL C01845 V=800.0 PL=0
MOVL C01846 V=800.0 PL=0
MOVL C01847 V=800.0 PL=0
MOVL C01848 V=800.0 PL=0
MOVL C01849 V=800.0 PL=0
MOVL C01850 V=800.0 PL=0
MOVL C01851 V=800.0 PL=0
MOVL C01852 V=800.0 PL=0
MOVL C01853 V=800.0 PL=0
MOVL C01854 V=800.0 PL=0
MOVL C01855 V=800.0 PL=0
MOVL C01856 V=800.0 PL=0
MOVL C01857 V=800.0 PL=0
MOVL C01858 V=800.0 PL=0
MOVL C01859 V=800.0 PL=0
MOVL C01860 V=800.0 PL=0
MOVL C01861 V=800.0 PL=0
MOVL C01862 V=800.0 PL=0
MOVL C01863 V=800.0 PL=0
MOVL C01864 V=800.0 PL=0
MOVL C01865 V=800.0 PL=0
MOVL C01866 V=800.0 PL=0
MOVL C01867 V=800.0 PL=0
MOVL C01868 V=800.0 PL=0
MOVL C01869 V=800.0 PL=0
MOVL C01870 V=800.0 PL=0
MOVL C01871 V=800.0 PL=0
MOVL C01872 V=800.0 PL=0
MOVL C01873 V=800.0 PL=0
MOVL C01874 V=800.0 PL=0
MOVL C01875 V=800.0 PL=0
MOVL C01876 V=800.0 PL=0
MOVL C01877 V=800.0 PL=0
MOVL C01878 V=800.0 PL=0
MOVL C01879 V=800.0 PL=0
MOVL C01880 V=800.0 PL=0
MOVL C01881 V=800.0 PL=0
MOVL C01882 V=800.0 PL=0
MOVL C01883 V=800.0 PL=0
MOVL C01884 V=800.0 PL=0
MOVL C01885 V=800.0 PL=0
MOVL C01886 V=800.0 PL=0
MOVL C01887 V=800.0 PL=0
MOVL C01888 V=800.0 PL=0
MOVL C01889 V=800.0 PL=0
MOVL C01890 V=800.0 PL=0
MOVL C01891 V=800.0 PL=0
MOVL C01892 V=800.0 PL=0
MOVL C01893 V=800.0 PL=0
MOVL C01894 V=800.0 PL=0
MOVL C01895 V=800.0 PL=0
MOVL C01896 V=800.0 PL=0
MOVL C01897 V=800.0 PL=0
MOVL C01898 V=800.0 PL=0
MOVL C01899 V=800.0 PL=0
MOVL C01900 V=800.0 PL=0
MOVL C01901 V=800.0 PL=0
MOVL C01902 V=800.0 PL=0
MOVL C01903 V=800.0 PL=0
MOVL C01904 V=800.0 PL=0
MOVL C01905 V=800.0 PL=0
MOVL C01906 V=800.0 PL=0
MOVL C01907 V=800.0 PL=0
MOVL C01908 V=800.0 PL=0
MOVL C01909 V=800.0 PL=0
MOVL C01910 V=800.0 PL=0
MOVL C01911 V=800.0 PL=0
MOVL C01912 V=800.0 PL=0
MOVL C01913 V=800.0 PL=0
MOVL C01914 V=800.0 PL=0
MOVL C01915 V=800.0 PL=0
MOVL C01916 V=800.0 PL=0
MOVL C01917 V=800.0 PL=0
MOVL C01918 V=800.0 PL=0
MOVL C01919 V=800.0 PL=0
MOVL C01920 V=800.0 PL=0
MOVL C01921 V=800.0 PL=0
MOVL C01922 V=800.0 PL=0
MOVL C01923 V=800.0 PL=0
MOVL C01924 V=800.0 PL=0
MOVL C01925 V=800.0 PL=0
MOVL C01926 V=800.0 PL=0
MOVL C01927 V=800.0 PL=0
MOVL C01928 V=800.0 PL=0
MOVL C01929 V=800.0 PL=0
MOVL C01930 V=800.0 PL=0
MOVL C01931 V=800.0 PL=0
MOVL C01932 V=800.0 PL=0
MOVL C01933 V=800.0 PL=0
MOVL C01934 V=800.0 PL=0
MOVL C01935 V=800.0 PL=0
MOVL C01936 V=800.0 PL=0
MOVL C01937 V=800.0 PL=0
MOVL C01938 V=800.0 PL=0
MOVL C01939 V=800.0 PL=0
MOVL C01940 V=800.0 PL=0
MOVL C01941 V=800.0 PL=0
MOVL C01942 V=800.0 PL=0
MOVL C01943 V=800.0 PL=0
MOVL C01944 V=800.0 PL=0
MOVL C01945 V=800.0 PL=0
MOVL C01946 V=800.0 PL=0
MOVL C01947 V=800.0 PL=0
MOVL C01948 V=800.0 PL=0
MOVL C01949 V=800.0 PL=0
MOVL C01950 V=800.0 PL=0
MOVL C01951 V=800.0 PL=0
MOVL C01952 V=800.0 PL=0
MOVL C01953 V=800.0 PL=0
MOVL C01954 V=800.0 PL=0
MOVL C01955 V=800.0 PL=0
MOVL C01956 V=800.0 PL=0
MOVL C01957 V=800.0 PL=0
MOVL C01958 V=800.0 PL=0
MOVL C01959 V=800.0 PL=0
MOVL C01960 V=800.0 PL=0
MOVL C01961 V=800.0 PL=0
MOVL C01962 V=800.0 PL=0
MOVL C01963 V=800.0 PL=0
MOVL C01964 V=800.0 PL=0
MOVL C01965 V=800.0 PL=0
MOVL C01966 V=800.0 PL=0
MOVL C01967 V=800.0 PL=0
MOVL C01968 V=800.0 PL=0
MOVL C01969 V=800.0 PL=0
MOVL C01970 V=800.0 PL=0
MOVL C01971 V=800.0 PL=0
MOVL C01972 V=800.0 PL=0
MOVL C01973 V=800.0 PL=0
MOVL C01974 V=800.0 PL=0
MOVL C01975 V=800.0 PL=0
MOVL C01976 V=800.0 PL=0
MOVL C01977 V=800.0 PL=0
MOVL C01978 V=800.0 PL=0
MOVL C01979 V=800.0 PL=0
MOVL C01980 V=800.0 PL=0
MOVL C01981 V=800.0 PL=0
MOVL C01982 V=800.0 PL=0
MOVL C01983 V=800.0 PL=0
MOVL C01984 V=800.0 PL=0
MOVL C01985 V=800.0 PL=0
MOVL C01986 V=800.0 PL=0
MOVL C01987 V=800.0 PL=0
MOVL C01988 V=800.0 PL=0
MOVL C01989 V=800.0 PL=0
MOVL C01990 V=800.0 PL=0
MOVL C01991 V=800.0 PL=0
MOVL C01992 V=800.0 PL=0
MOVL C01993 V=800.0 PL=0
MOVL C01994 V=800.0 PL=0
MOVL C01995 V=800.0 PL=0
MOVL C01996 V=800.0 PL=0
MOVL C01997 V=800.0 PL=0
MOVL C01998 V=800.0 PL=0
MOVL C01999 V=800.0 PL=0
MOVL C02000 V=800.0 PL=0
MOVL C02001 V=800.0 PL=0
MOVL C02002 V=800.0 PL=0
MOVL C02003 V=800.0 PL=0
MOVL C02004 V=800.0 PL=0
MOVL C02005 V=800.0 PL=0
MOVL C02006 V=800.0 PL=0
MOVL C02007 V=800.0 PL=0
MOVL C02008 V=800.0 PL=0
MOVL C02009 V=800.0 PL=0
MOVL C02010 V=800.0 PL=0
MOVL C02011 V=800.0 PL=0
MOVL C02012 V=800.0 PL=0
MOVL C02013 V=800.0 PL=0
MOVL C02014 V=800.0 PL=0
MOVL C02015 V=800.0 PL=0
MOVL C02016 V=800.0 PL=0
MOVL C02017 V=800.0 PL=0
MOVL C02018 V=800.0 PL=0
MOVL C02019 V=800.0 PL=0
MOVL C02020 V=800.0 PL=0
MOVL C02021 V=800.0 PL=0
MOVL C02022 V=800.0 PL=0
MOVL C02023 V=800.0 PL=0
MOVL C02024 V=800.0 PL=0
MOVL C02025 V=800.0 PL=0
MOVL C02026 V=800.0 PL=0
MOVL C02027 V=800.0 PL=0
MOVL C02028 V=800.0 PL=0
MOVL C02029 V=800.0 PL=0
MOVL C02030 V=800.0 PL=0
MOVL C02031 V=800.0 PL=0
MOVL C02032 V=800.0 PL=0
MOVL C02033 V=800.0 PL=0
MOVL C02034 V=800.0 PL=0
MOVL C02035 V=800.0 PL=0
MOVL C02036 V=800.0 PL=0
MOVL C02037 V=800.0 PL=0
MOVL C02038 V=800.0 PL=0
MOVL C02039 V=800.0 PL=0
MOVL C02040 V=800.0 PL=0
MOVL C02041 V=800.0 PL=0
MOVL C02042 V=800.0 PL=0
MOVL C02043 V=800.0 PL=0
MOVL C02044 V=800.0 PL=0
MOVL C02045 V=800.0 PL=0
MOVL C02046 V=800.0 PL=0
MOVL C02047 V=800.0 PL=0
MOVL C02048 V=800.0 PL=0
MOVL C02049 V=800.0 PL=0
MOVL C02050 V=800.0 PL=0
MOVL C02051 V=800.0 PL=0
MOVL C02052 V=800.0 PL=0
MOVL C02053 V=800.0 PL=0
MOVL C02054 V=800.0 PL=0
MOVL C02055 V=800.0 PL=0
MOVL C02056 V=800.0 PL=0
MOVL C02057 V=800.0 PL=0
MOVL C02058 V=800.0 PL=0
MOVL C02059 V=800.0 PL=0
MOVL C02060 V=800.0 PL=0
MOVL C02061 V=800.0 PL=0
MOVL C02062 V=800.0 PL=0
MOVL C02063 V=800.0 PL=0
MOVL C02064 V=800.0 PL=0
MOVL C02065 V=800.0 PL=0
MOVL C02066 V=800.0 PL=0
MOVL C02067 V=800.0 PL=0
MOVL C02068 V=800.0 PL=0
MOVL C02069 V=800.0 PL=0
MOVL C02070 V=800.0 PL=0
MOVL C02071 V=800.0 PL=0
MOVL C02072 V=800.0 PL=0
MOVL C02073 V=800.0 PL=0
MOVL C02074 V=800.0 PL=0
MOVL C02075 V=800.0 PL=0
MOVL C02076 V=800.0 PL=0
MOVL C02077 V=800.0 PL=0
MOVL C02078 V=800.0 PL=0
MOVL C02079 V=800.0 PL=0
MOVL C02080 V=800.0 PL=0
MOVL C02081 V=800.0 PL=0
MOVL C02082 V=800.0 PL=0
MOVL C02083 V=800.0 PL=0
MOVL C02084 V=800.0 PL=0
MOVL C02085 V=800.0 PL=0
MOVL C02086 V=800.0 PL=0
MOVL C02087 V=800.0 PL=0
MOVL C02088 V=800.0 PL=0
MOVL C02089 V=800.0 PL=0
MOVL C02090 V=800.0 PL=0
MOVL C02091 V=800.0 PL=0
MOVL C02092 V=800.0 PL=0
MOVL C02093 V=800.0 PL=0
MOVL C02094 V=800.0 PL=0
MOVL C02095 V=800.0 PL=0
MOVL C02096 V=800.0 PL=0
MOVL C02097 V=800.0 PL=0
MOVL C02098 V=800.0 PL=0
MOVL C02099 V=800.0 PL=0
MOVL C02100 V=800.0 PL=0
MOVL C02101 V=800.0 PL=0
MOVL C02102 V=800.0 PL=0
MOVL C02103 V=800.0 PL=0
MOVL C02104 V=800.0 PL=0
MOVL C02105 V=800.0 PL=0
MOVL C02106 V=800.0 PL=0
MOVL C02107 V=800.0 PL=0
MOVL C02108 V=800.0 PL=0
MOVL C02109 V=800.0 PL=0
MOVL C02110 V=800.0 PL=0
MOVL C02111 V=800.0 PL=0
MOVL C02112 V=800.0 PL=0
MOVL C02113 V=800.0 PL=0
MOVL C02114 V=800.0 PL=0
MOVL C02115 V=800.0 PL=0
MOVL C02116 V=800.0 PL=0
MOVL C02117 V=800.0 PL=0
MOVL C02118 V=800.0 PL=0
MOVL C02119 V=800.0 PL=0
MOVL C02120 V=800.0 PL=0
MOVL C02121 V=800.0 PL=0
MOVL C02122 V=800.0 PL=0
MOVL C02123 V=800.0 PL=0
MOVL C02124 V=800.0 PL=0
MOVL C02125 V=800.0 PL=0
MOVL C02126 V=800.0 PL=0
MOVL C02127 V=800.0 PL=0
MOVL C02128 V=800.0 PL=0
MOVL C02129 V=800.0 PL=0
MOVL C02130 V=800.0 PL=0
MOVL C02131 V=800.0 PL=0
MOVL C02132 V=800.0 PL=0
MOVL C02133 V=800.0 PL=0
MOVL C02134 V=800.0 PL=0
MOVL C02135 V=800.0 PL=0
MOVL C02136 V=800.0 PL=0
MOVL C02137 V=800.0 PL=0
MOVL C02138 V=800.0 PL=0
